//bReadyToRead :=  Tc2_System.MEMCMP( ADR( stTimeStamp), ADR (stNullTimeStamp), SIZEOF(stTimeStamp)) <> 0 AND NOT  fbGetSystemTime.BUSY;	
			(*keczi*)	(*zrobione po to zeby w wypadku jak po starcie PLC na HMI mial pokazywac czas alarmu '00:00:00', zebyb poczekal az faktycznie pokazuje date i czas*)

//Get Current System Time
fbGetSystemTime(NETID := ,
				START := bFirstScan OR bUpdateSysTime,
				TMOUT := ,
				BUSY => ,
				ERR => ,
				ERRID => ,
				TIMESTR => );
				
//Get system time done detection - one-shot
rtrigSysTimeCollected(CLK := NOT fbGetSystemTime.BUSY);

//Synchronize Real-Time clock with system time
fbRTClock(	EN := rtrigSysTimeCollected.Q, 
			PDT := fbGetSystemTime.TIMESTR,
			CDT => stTimeStamp, 
			Q => bReadyToRead);

// System Date and Time in Proper Order 
IF bReadyToRead THEN
	sRawDateTime := SYSTEMTIME_TO_STRING(stTimeStamp);  // format: YYYY-MM-DD-hh:mm:ss.xxx
	GVL_HMI_GLOBAL.sSystemDate := CONCAT(CONCAT(CONCAT(CONCAT(MID(sRawDateTime, 2, 9), '.'),  MID(sRawDateTime, 2, 6)), '.'), LEFT(sRawDateTime, 4));
	GVL_HMI_GLOBAL.sSystemTime := MID(sRawDateTime, 8, 12);
	sDateTime := CONCAT(CONCAT(GVL_HMI_GLOBAL.sSystemDate, '  '), GVL_HMI_GLOBAL.sSystemTime);
	sDateTimeSpaces	:= CONCAT(sDateTime, '    ');
END_IF;

bFirstScan := FALSE;
END_ACTION

END_PROGRAM

// ---- POUs/A_Master/PRG_MasterSystemTime.TcPOU
PROGRAM PRG_MasterSystemTime
VAR
	//Variables
	bReadyToRead				:BOOL;
	bFirstScan					:BOOL := TRUE;
	bUpdateSysTime				:BOOL; //Output of pulse generator
	tSysTimeUpdatePeriod		:TIME := T#5S;
	stTimeStamp					:TIMESTRUCT;
	stNullTimeStamp				:TIMESTRUCT;
	sRawDateTime				:STRING;
	sSystemDate					:STRING;
	sSystemTime					:STRING;
	sDateTime					:STRING;
	sDateTimeSpaces				:STRING;
	
	stTimeTest                  :TIMESTRUCT;
	sttimeTest2                 :TIMESTRUCT;
	sTestTime                   :STRING;
	nSectTest                   :DINT;
	bStartTest                  :BOOL;
	bStsrtTest2                 :BOOL;
	
	
	//Functions
	fbGetSystemTime				:TC2_Utilities.NT_GetTime;
	fbRTClock					:TC2_Utilities.RTC_EX2;		//Local real-time clock
	tonTimeUpdateGen			:TC2_Utilities.TON;			//Pulse generator for triggering fbGetSystemTime function
	rtrigSysTimeCollected		:TC2_Utilities.R_TRIG;		//System time collected

    fbTimerControl              :FB_TimeControl;
	bStartTimeTest              :BOOL;
	bResetTimeTest              :BOOL;
	nTimeHourTest               :DINT;
	nTimeMinTest                :DINT;
	nTimeSecTest                :DINT;
	nTimeTotalSecTest           :DINT;
END_VAR

//Aux functions call
tonTimeUpdateGen(	IN := NOT bUpdateSysTime,
					PT := tSysTimeUpdatePeriod,
					Q => bUpdateSysTime);

//bReadyToRead :=  Tc2_System.MEMCMP( ADR( stTimeStamp), ADR (stNullTimeStamp), SIZEOF(stTimeStamp)) <> 0 AND NOT  fbGetSystemTime.BUSY;	
			(*keczi*)	(*zrobione po to zeby w wypadku jak po starcie PLC na HMI mial pokazywac czas alarmu '00:00:00', zebyb poczekal az faktycznie pokazuje date i czas*)

//Get Current System Time
fbGetSystemTime(NETID := ,
				START := bFirstScan OR bUpdateSysTime,
				TMOUT := ,
				BUSY => ,
				ERR => ,
				ERRID => ,
				TIMESTR => );
				
//Get system time done detection - one-shot
rtrigSysTimeCollected(CLK := NOT fbGetSystemTime.BUSY);

//Synchronize Real-Time clock with system time
fbRTClock(	EN := rtrigSysTimeCollected.Q, 
			PDT := fbGetSystemTime.TIMESTR,
			CDT => stTimeStamp, 
			Q => bReadyToRead);

// System Date and Time in Proper Order 
IF bReadyToRead THEN
	sRawDateTime := SYSTEMTIME_TO_STRING(stTimeStamp);  // format: YYYY-MM-DD-hh:mm:ss.xxx
	sSystemDate := CONCAT(CONCAT(CONCAT(CONCAT(MID(sRawDateTime, 2, 9), '.'),  MID(sRawDateTime, 2, 6)), '.'), LEFT(sRawDateTime, 4));
	sSystemTime := MID(sRawDateTime, 8, 12);
	sDateTime := CONCAT(CONCAT(sSystemDate, '  '), sSystemTime);
	sDateTimeSpaces	:= CONCAT(sDateTime, '    ');
	
	//Time to write to CSV Files
	//nSystemTime := sSystemTime;
END_IF;

bFirstScan := FALSE;

IF bStartTest THEN
	sTestTime:= SYSTEMTIME_TO_STRING(stTimeTest);
END_IF

fbTimerControl( bEnable  :=  bStartTimeTest,
	            bReset   :=  bResetTimeTest,
				nHour     => nTimeHourTest,
				nMin      => nTimeMinTest,
				nSec      => nTimeSecTest,
				nTotalSec => nTimeTotalSecTest );

END_PROGRAM

// ---- POUs/E_HMI/PRG_HMI.TcPOU
PROGRAM PRG_HMI
VAR
	

	tonCaseDelay				: ARRAY [1..20] OF TON;
	tofCase						: ARRAY [1..20] OF TOF;
	rtrigCaseTriger				: ARRAY [1..20] OF R_TRIG;
	nHeightMeasureStateValue	: ARRAY [1..4] OF INT;
	i							: INT;

END_VAR

ACT_ScreensNamesSet();
ACT_Buttons();
ACT_TimTrig();
ACT_General();

ACTION ACT_Buttons:
ACT_TimTrig();

IF tonCaseDelay[1].Q THEN
	
		GVL_HMI_GLOBAL.bResetButton	:= FALSE;
		
END_IF
IF tonCaseDelay[2].Q THEN
	
		GVL_HMI_GLOBAL.bStopButton	:= FALSE;
		
END_IF
IF tonCaseDelay[3].Q THEN
	
		GVL_HMI_GLOBAL.bStartButton	:= FALSE;
		
END_IF

IF GVL_HMI_GLOBAL.bStartLeakMan THEN
	GVL_IO.dw_B07_i28General_I_O.bStart := TRUE;
END_IF
IF tonCaseDelay[4].Q THEN
	
		GVL_HMI_GLOBAL.bStartLeakMan	:= FALSE;
		GVL_IO.dw_B07_i28General_I_O.bStart := FALSE;
END_IF

IF GVL_HMI_GLOBAL.bStopLeakMan THEN
	GVL_IO.dw_B07_i28General_I_O.bStop := TRUE;
END_IF
IF tonCaseDelay[5].Q THEN
	
		GVL_HMI_GLOBAL.bStopLeakMan	:= FALSE;
		GVL_IO.dw_B07_i28General_I_O.bStop := FALSE;
		
END_IF

IF GVL_HMI_GLOBAL.bResetLeakMan THEN
	GVL_IO.dw_B07_i28General_I_O.bReset := TRUE;
END_IF
IF tonCaseDelay[6].Q THEN
	
		GVL_HMI_GLOBAL.bResetLeakMan	:= FALSE;
		GVL_IO.dw_B07_i28General_I_O.bReset := FALSE;
		
END_IF

IF tonCaseDelay[7].Q THEN
	
		GVL_HMI_GLOBAL.bShutDown	:= FALSE;
		
END_IF
IF tonCaseDelay[8].Q THEN
	
		GVL_HMI_GLOBAL.bSetLeakProgramID	:= FALSE;
		
END_IF

// Stopper Press Enable/Disable Message

IF GVL_HMI_GLOBAL.bStopperPressEnable THEN 
	GVL_HMI_GLOBAL.sStopperEnableDisable:='STOPPER PRESS ENABLED';
	ELSE
	GVL_HMI_GLOBAL.sStopperEnableDisable:='STOPPER PRESS DISABLED';
END_IF
END_ACTION

ACTION ACT_General:
IF  tofCase[1].Q
	AND (NOT GVL_MASTER.stMasterControl.bNoMachineImmediateFault OR NOT GVL_MASTER.stMasterControl.bNoCycleStopFault) THEN
	GVL_HMI_GLOBAL.bAutoCycleFaultDialog := TRUE;
END_IF
END_ACTION

ACTION ACT_ScreensNamesSet:
GVL_HMI_GLOBAL.aIOScreen[0] := 'Overview';
GVL_HMI_GLOBAL.aIOScreen[1] := 'HMI - CP2913-0000 | Beckhoff HMI';
GVL_HMI_GLOBAL.aIOScreen[2] := 'PLC - C6015-0010 | Beckhoff PLC | Windows 10 Embedded';
GVL_HMI_GLOBAL.aIOScreen[3] := 'Terminal 1- EK1100 | EtherCAT Coupler';
GVL_HMI_GLOBAL.aIOScreen[4] := 'Terminal 2 - EL6070 | Licence ';
GVL_HMI_GLOBAL.aIOScreen[5] := CONCAT('Terminal 3 - ' , GVL_IO.dw_T02_EL1809.sTerminalName);
GVL_HMI_GLOBAL.aIOScreen[6] := CONCAT('Terminal 4 - ' , GVL_IO.dw_T03_EL2809.sTerminalName);
GVL_HMI_GLOBAL.aIOScreen[7] := 'Terminal 12 - EL6631 |  2-port communication interface';
GVL_HMI_GLOBAL.aIOScreen[8] := 'I28 | Cincinnati Leak Tester | ProfiNET';

GVL_HMI_GLOBAL.aManualScreen[0] := 'Cognex | Vision Test';
GVL_HMI_GLOBAL.aManualScreen[1] := 'Keyence | Height Test';
GVL_HMI_GLOBAL.aManualScreen[2] := 'Cincinnati | Leak Test';
END_ACTION

ACTION ACT_TimTrig:


tonCaseDelay[1](IN:= GVL_HMI_GLOBAL.bResetButton,PT:=T#500MS);
tonCaseDelay[2](IN:= GVL_HMI_GLOBAL.bStopButton,PT:=T#500MS);
tonCaseDelay[3](IN:= GVL_HMI_GLOBAL.bStartButton,PT:=T#500MS);
tonCaseDelay[4](IN:= GVL_HMI_GLOBAL.bStartLeakMan,PT:=T#500MS);
tonCaseDelay[5](IN:= GVL_HMI_GLOBAL.bStopLeakMan,PT:=T#500MS);
tonCaseDelay[6](IN:= GVL_HMI_GLOBAL.bResetLeakMan,PT:=T#500MS);
//tonCaseDelay[7](IN:= GVL_HMI_GLOBAL.bShutDown,PT:=T#500MS);
tonCaseDelay[8](IN:= GVL_HMI_GLOBAL.bSetLeakProgramID,PT:=T#5S);
tonCaseDelay[9](IN:= ,PT:=T#1S);
tonCaseDelay[10](IN:= ,PT:=T#1S);

tofCase[1](IN:= GVL_MASTER.stStationSruct[0].nState > 1000 AND GVL_MASTER.stStationSruct[0].nState < 1900,PT:=T#1S);



rtrigCaseTriger[1](CLK := GVL_MASTER.stNest.bPieceReject);
END_ACTION

END_PROGRAM

// ---- POUs/G_Utility/PRG_Puls.TcPOU
PROGRAM PRG_Puls
VAR
    //=== Master Pulses ===//
	fbScalingFlash  :FB_Pulse;
	fbScalingFlash4 :FB_Pulse;
	fbScalingFlash5 :FB_Pulse;
	fbFlash100Hz    :FB_Pulse;
	fbFlash10Hz		:FB_Pulse;
	fbFlash10HzB    :FB_Pulse;
	fbFlash4Hz		:FB_Pulse;
	fbFlash2Hz		:FB_Pulse;
	fbFlash1Hz		:FB_Pulse;			

END_VAR

    //=== Master Pulses ===//
(**************************************************************************************************)
fbScalingFlash(
	bEnable	:=	TRUE,
	tPulseOn	:=	T#2MS,
	tPulseOff	:=	T#2MS,
	bFlash		=>	GVL_MASTER.bFlashScale
);

fbScalingFlash4(
     bEnable	:=	TRUE,
	tPulseOn	:=	T#4MS,
	tPulseOff	:=	T#4MS,
	bFlash		=>	GVL_MASTER.bFlashScale4
);
fbScalingFlash5(
     bEnable	:=	TRUE,
	tPulseOn	:=	T#5MS,
	tPulseOff	:=	T#5MS,
	bFlash		=>	GVL_MASTER.bFlashScale5
);



fbFlash100Hz(
	bEnable	:=	TRUE,
	tPulseOn	:=	T#10MS,
	tPulseOff	:=	T#10MS,
	bFlash		=>	GVL_MASTER.bFlash100Hz
);


fbFlash10HzB ( 
    bEnable	    :=	TRUE,
	tPulseOn	:=	T#20MS,//  T#50MS,
	tPulseOff	:=	T#20MS,//  T#50MS,
	bFlash		=>	GVL_MASTER.bFlash10BHz
);


fbFlash10Hz(
	bEnable	:=	TRUE,
	tPulseOn	:=	T#100MS,
	tPulseOff	:=	T#100MS,
	bFlash		=>	GVL_MASTER.bFlash10Hz
);


fbFlash4Hz(
	bEnable	:=	TRUE,
	tPulseOn	:=	T#250MS,
	tPulseOff	:=	T#250MS,
	bFlash		=>	GVL_MASTER.bFlash4Hz
);

fbFlash2Hz(
	bEnable	:=	TRUE,
	tPulseOn	:=	T#500MS,
	tPulseOff	:=	T#500MS,
	bFlash		=>	GVL_MASTER.bFlash2Hz
);

fbFlash1Hz(
	bEnable	:=	TRUE,
	tPulseOn	:=	T#1000MS,
	tPulseOff	:=	T#1000MS,
	bFlash		=>	GVL_MASTER.bFlash1Hz
);

END_PROGRAM

// ---- POUs/A_Master/PRG_TerminBoxInfo.TcPOU
PROGRAM PRG_TerminBoxInfo
VAR
END_VAR

//Terminal 0
GVL_IO.dwTerminalInfo[1].fbTerminalInfo(nTerminalState:= 8,
                                        sTerminalState => GVL_IO.dwTerminalInfo[0].sTerminalInfo);
//Terminal 1
GVL_IO.dwTerminalInfo[1].fbTerminalInfo(nTerminalState:= GVL_IO.dwTerminalInfo[1].nTerminal_State,
                                        sTerminalState => GVL_IO.dwTerminalInfo[1].sTerminalInfo);  
//Terminal 2
GVL_IO.dwTerminalInfo[2].fbTerminalInfo(nTerminalState:= GVL_IO.dwTerminalInfo[2].nTerminal_State,
                                        sTerminalState => GVL_IO.dwTerminalInfo[2].sTerminalInfo); 
//Terminal 3
GVL_IO.dwTerminalInfo[3].fbTerminalInfo(nTerminalState:= GVL_IO.dwTerminalInfo[3].nTerminal_State,
                                        sTerminalState => GVL_IO.dwTerminalInfo[3].sTerminalInfo); 
//Terminal 4
GVL_IO.dwTerminalInfo[4].fbTerminalInfo(nTerminalState:= GVL_IO.dwTerminalInfo[4].nTerminal_State,
                                        sTerminalState => GVL_IO.dwTerminalInfo[4].sTerminalInfo); 
//Terminal 5
GVL_IO.dwTerminalInfo[5].fbTerminalInfo(nTerminalState:= GVL_IO.dwTerminalInfo[5].nTerminal_State,
                                        sTerminalState => GVL_IO.dwTerminalInfo[5].sTerminalInfo); 
//Terminal 6
GVL_IO.dwTerminalInfo[6].fbTerminalInfo(nTerminalState:= GVL_IO.dwTerminalInfo[6].nTerminal_State,
                                        sTerminalState => GVL_IO.dwTerminalInfo[6].sTerminalInfo); 
//Terminal 7
GVL_IO.dwTerminalInfo[7].fbTerminalInfo(nTerminalState:= GVL_IO.dwTerminalInfo[7].nTerminal_State,
                                        sTerminalState => GVL_IO.dwTerminalInfo[7].sTerminalInfo); 
//Terminal 8
GVL_IO.dwTerminalInfo[8].fbTerminalInfo(nTerminalState:= GVL_IO.dwTerminalInfo[8].nTerminal_State,
                                        sTerminalState => GVL_IO.dwTerminalInfo[8].sTerminalInfo); 
//Terminal 9
GVL_IO.dwTerminalInfo[9].fbTerminalInfo(nTerminalState:= GVL_IO.dwTerminalInfo[9].nTerminal_State,
                                        sTerminalState => GVL_IO.dwTerminalInfo[9].sTerminalInfo); 
//Terminal 10
GVL_IO.dwTerminalInfo[10].fbTerminalInfo(nTerminalState:= GVL_IO.dwTerminalInfo[10].nTerminal_State,
                                        sTerminalState => GVL_IO.dwTerminalInfo[10].sTerminalInfo); 
//Terminal 11
GVL_IO.dwTerminalInfo[11].fbTerminalInfo(nTerminalState:= GVL_IO.dwTerminalInfo[11].nTerminal_State,
                                        sTerminalState => GVL_IO.dwTerminalInfo[11].sTerminalInfo); 
//Terminal 12
GVL_IO.dwTerminalInfo[12].fbTerminalInfo(nTerminalState:= GVL_IO.dwTerminalInfo[12].nTerminal_State,
                                        sTerminalState => GVL_IO.dwTerminalInfo[12].sTerminalInfo); 										
//Terminal 13
GVL_IO.dwTerminalInfo[13].fbTerminalInfo(nTerminalState:= GVL_IO.dwTerminalInfo[13].nTerminal_State,
                                        sTerminalState => GVL_IO.dwTerminalInfo[13].sTerminalInfo); 
//Terminal 14
GVL_IO.dwTerminalInfo[14].fbTerminalInfo(nTerminalState:= GVL_IO.dwTerminalInfo[14].nTerminal_State,
                                        sTerminalState => GVL_IO.dwTerminalInfo[14].sTerminalInfo);
										
//Terminal 15
GVL_IO.dwTerminalInfo[15].fbTerminalInfo(nTerminalState:= GVL_IO.dwTerminalInfo[15].nTerminal_State,
                                        sTerminalState => GVL_IO.dwTerminalInfo[15].sTerminalInfo); 
//Terminal 16
GVL_IO.dwTerminalInfo[16].fbTerminalInfo(nTerminalState:= 8,
                                        sTerminalState => GVL_IO.dwTerminalInfo[16].sTerminalInfo);										

//Terminal 17
GVL_IO.dwTerminalInfo[17].fbTerminalInfo(nTerminalState:= 8,
                                        sTerminalState => GVL_IO.dwTerminalInfo[17].sTerminalInfo);

//Terminal 18
GVL_IO.dwTerminalInfo[18].fbTerminalInfo(nTerminalState:= 8,
                                        sTerminalState => GVL_IO.dwTerminalInfo[18].sTerminalInfo);

//Terminal 19
GVL_IO.dwTerminalInfo[19].fbTerminalInfo(nTerminalState:= 8,
                                        sTerminalState => GVL_IO.dwTerminalInfo[19].sTerminalInfo);

//Terminal 20
GVL_IO.dwTerminalInfo[20].fbTerminalInfo(nTerminalState:= 8,
                                        sTerminalState => GVL_IO.dwTerminalInfo[20].sTerminalInfo);
																				
// Box 15
GVL_IO.dwBoxInfo[15].fbBoxInfo(nPnIoBoxState := GVL_IO.dwBoxInfo[15].nPnIoBoxState,    	
                               nPnIoBoxDiag  := GVL_IO.dwBoxInfo[15].nPnIoBoxDiag,
							   sBoxState      => GVL_IO.dwBoxInfo[15].sBoxState,
                               sBoxDiag       => GVL_IO.dwBoxInfo[15].sBoxDiag);
							   
//===========================================================================================================

END_PROGRAM

// ---- POUs/C_LeakTest/PRG_LeakTestEvents_Info.TcPOU
PROGRAM PRG_LeakTestEvents_Info
VAR
	
	asLeakTesterSegments 				: ARRAY [0..200] OF WSTRING;
	asLeakTesterTestData 				: ARRAY [0..200] OF WSTRING;
	asLeakTesterUnit 	 				: ARRAY [0..200] OF WSTRING;
	asLeakTesterPrecision				: ARRAY [0..10]  OF WSTRING;
	asLeakTesterProgramEvaluation		: ARRAY [0..20]  OF WSTRING;
	asLeakTesterTestEvaluation			: ARRAY [0..150]  OF WSTRING;
	asLeakTesterTestType				: ARRAY [0..25]  OF WSTRING;
	fLeakTesterActive					: F_TRIG;
	bLeakTesterActive					: BOOL;
	Test1								: BOOL;
		
	i									: DINT;
	

END_VAR

ACT_LiveSegmentCode();
ACT_LeakTesterTestData();
ACT_LeakTesterUnit();
ACT_Precision();
ACT_ProgramEvaluation();
ACT_LeakTesterTestEvaluation();
ACT_TestType();

//Last Result DATA

GVL_IO.dw_B07_i28LastResult.sPartEvaluation 		:= asLeakTesterTestData[GVL_IO.dw_B07_i28LastResult.inTestType];
GVL_IO.dw_B07_i28LastResult.sPrecision				:= asLeakTesterPrecision[GVL_IO.dw_B07_i28LastResult.inPrecisionCode];
GVL_IO.dw_B07_i28LastResult.sTestType				:= asLeakTesterTestType[ GVL_IO.dw_B07_i28LastResult.inPartEvaluation];
GVL_IO.dw_B07_i28LastResult.sUnit1      			:= asLeakTesterUnit[GVL_IO.dw_B07_i28LastResult.inUnitCode1];
GVL_IO.dw_B07_i28LastResult.sUnit2					:= asLeakTesterUnit[GVL_IO.dw_B07_i28LastResult.inUnitCode2];
GVL_IO.dw_B07_i28LastResult.sVariable1				:= asLeakTesterTestData[GVL_IO.dw_B07_i28LastResult.inVariableCode1];
GVL_IO.dw_B07_i28LastResult.sVariable2				:= asLeakTesterTestData[GVL_IO.dw_B07_i28LastResult.inVariableCode2];

//Live DATA


GVL_IO.dw_B07_i28LiveMeasurement.sPrecision1		:= asLeakTesterPrecision[GVL_IO.dw_B07_i28LiveMeasurement.inPrecisionCode1];
GVL_IO.dw_B07_i28LiveMeasurement.sPrecision2		:= asLeakTesterPrecision[GVL_IO.dw_B07_i28LiveMeasurement.inPrecisionCode2];
GVL_IO.dw_B07_i28LiveMeasurement.sPrecision3		:= asLeakTesterPrecision[GVL_IO.dw_B07_i28LiveMeasurement.inPrecisionCode3];
GVL_IO.dw_B07_i28LiveMeasurement.sPrecision4		:= asLeakTesterPrecision[GVL_IO.dw_B07_i28LiveMeasurement.inPrecisionCode4];
GVL_IO.dw_B07_i28LiveMeasurement.sSegmentCode		:= asLeakTesterSegments[GVL_IO.dw_B07_i28LiveMeasurement.inSegmentCode];
GVL_IO.dw_B07_i28LiveMeasurement.sUnit1				:= asLeakTesterUnit[GVL_IO.dw_B07_i28LiveMeasureMENT.inUnitCode1];
GVL_IO.dw_B07_i28LiveMeasurement.sUnit2				:= asLeakTesterUnit[GVL_IO.dw_B07_i28LiveMeasureMENT.inUnitCode2];
GVL_IO.dw_B07_i28LiveMeasurement.sUnit3				:= asLeakTesterUnit[GVL_IO.dw_B07_i28LiveMeasureMENT.inUnitCode3];
GVL_IO.dw_B07_i28LiveMeasurement.sUnit4				:= asLeakTesterUnit[GVL_IO.dw_B07_i28LiveMeasureMENT.inUnitCode4];
GVL_IO.dw_B07_i28LiveMeasurement.sVariable1			:= asLeakTesterTestData[GVL_IO.dw_B07_i28LiveMeasurement.inVariableCode1];
GVL_IO.dw_B07_i28LiveMeasurement.sVariable2			:= asLeakTesterTestData[GVL_IO.dw_B07_i28LiveMeasurement.inVariableCode2];
GVL_IO.dw_B07_i28LiveMeasurement.sVariable3			:= asLeakTesterTestData[GVL_IO.dw_B07_i28LiveMeasurement.inVariableCode3];
GVL_IO.dw_B07_i28LiveMeasurement.sVariable4			:= asLeakTesterTestData[GVL_IO.dw_B07_i28LiveMeasurement.inVariableCode4];


ACT_LastResultSet();

ACTION ACT_LastResultSet:

fLeakTesterActive(CLK := GVL_IO.dw_B07_i28General_I_O.bTestActiveLiveData, Q => bLeakTesterActive);


IF bLeakTesterActive THEN
	
	FOR i :=200 TO 1 BY (-1) DO
		GVL_PERSIST.ast_i28LasResult[i]	:= GVL_PERSIST.ast_i28LasResult[i-1];
	END_FOR
	
	GVL_PERSIST.ast_i28LasResult[0] := GVL_IO.dw_B07_i28LastResult;
	GVL_PERSIST.ast_i28LasResult[0].sTime := GVL_HMI_GLOBAL.sSystemTime;
	GVL_PERSIST.ast_i28LasResult[0].sDate := GVL_HMI_GLOBAL.sSystemDate;

END_IF
END_ACTION

ACTION ACT_LeakTesterTestData:
asLeakTesterTestData[0] := "NO DATA";
asLeakTesterTestData[1] := "Elapsed Timer";
asLeakTesterTestData[2] := "Segment Timer";
asLeakTesterTestData[3] := "Test Execution Time";
asLeakTesterTestData[4] := "Target Pressure";
asLeakTesterTestData[5] := "Test Pressure";
asLeakTesterTestData[6] := "Master Part Profile Test Pressure";
asLeakTesterTestData[7] := "Master Part & Leak Profile Test Pressure";
asLeakTesterTestData[8] := "Leak Standard Calibrated Pressure";
asLeakTesterTestData[9] := "Self Test Pressure";
asLeakTesterTestData[10] := "Measured Pressure";
asLeakTesterTestData[11] := "Instrument Pressure";
asLeakTesterTestData[12] := "Master Gauge Pressure";
asLeakTesterTestData[13] := "Master Part Pressure Loss (Corrected)";
asLeakTesterTestData[14] := "Low Limit Pressure Loss";
asLeakTesterTestData[15] := "High Limit Pressure Loss";
asLeakTesterTestData[16] := "Master Part & Leak Pressure Loss (Corrected)";
asLeakTesterTestData[17] := "Pressure Loss (Corrected)";
asLeakTesterTestData[18] := "Pressure Loss (Actual Read)";
asLeakTesterTestData[19] := "Master Part Flow Offset (Corrected)";
asLeakTesterTestData[20] := "Performance Factor";
asLeakTesterTestData[21] := "Low Limit Rate";
asLeakTesterTestData[22] := "High Limit Rate";
asLeakTesterTestData[23] := "Loss Rate (Corrected)";
asLeakTesterTestData[24] := "Loss Rate (Actual Read)";
asLeakTesterTestData[25] := "Quik Test Pressure";
asLeakTesterTestData[26] := "Quik Test Loss (Corrected)";
asLeakTesterTestData[27] := "Quik Test Flow (Corrected)";
asLeakTesterTestData[28] := "Low Limit Leak Rate";
asLeakTesterTestData[29] := "High Limit Leak Rate";
asLeakTesterTestData[30] := "Predicted Leak Rate";
asLeakTesterTestData[31] := "Leak Rate";
asLeakTesterTestData[32] := "Corrected Leak Standard Calibrated Flow";
asLeakTesterTestData[33] := "Measured Flow";
asLeakTesterTestData[34] := "Environmental Drift Correction Offset";
asLeakTesterTestData[35] := "Transducer Type";
asLeakTesterTestData[36] := "Transducer Typical Residual";
asLeakTesterTestData[37] := "Transducer Zero Low Window";
asLeakTesterTestData[38] := "Transducer Zero High Window";
asLeakTesterTestData[39] := "Regulator Type";
asLeakTesterTestData[40] := "Analog A/D Value";
asLeakTesterTestData[41] := "Peak Pressure";
asLeakTesterTestData[42] := "Analog Input";
asLeakTesterTestData[43] := "Analog Output";
asLeakTesterTestData[44] := "Event Delta Pressure";
asLeakTesterTestData[45] := "Alternate Leak Rate";
asLeakTesterTestData[46] := "DP Master Part Pressure Loss (Corrected)";
asLeakTesterTestData[47] := "DP Master Part & Leak Pressure Loss (Corrected)";
asLeakTesterTestData[48] := "Master Part Quik Pressure Loss (Corrected)";
asLeakTesterTestData[49] := "Master Part Quik Pressure Loss (Actual Read)";
asLeakTesterTestData[50] := "Master Part & Leak Quik Pressure Loss (Corrected)";
asLeakTesterTestData[51] := "Master Part & Leak Quik Pressure Loss (Actual Read)";
asLeakTesterTestData[52] := "Master Part Quik Test Pressure";
asLeakTesterTestData[53] := "Master Part & Leak Quik Test Pressure";
asLeakTesterTestData[54] := "Master Part Quik DP Pressure Loss (Corrected)";
asLeakTesterTestData[55] := "Master Part Quik DP Pressure Loss (Actual Read)";
asLeakTesterTestData[56] := "Master Part & Leak Quik DP Pressure Loss (Actual Read)";
asLeakTesterTestData[57] := "Signal to Noise Ratio";
asLeakTesterTestData[58] := "Effective Number of Bits";
asLeakTesterTestData[59] := "Flicker Free Number of Bits";
asLeakTesterTestData[60] := "High Limit Percent Volume";
asLeakTesterTestData[61] := "Part Percent Volume";
asLeakTesterTestData[62] := "Reference Pressure";
asLeakTesterTestData[63] := "Fill Pressure";
asLeakTesterTestData[64] := "Transducer Cal/Verify - Number of Points";
asLeakTesterTestData[65] := "Transducer - Setpoint Pressure Value";
asLeakTesterTestData[66] := "Transducer - Instrument Pressure Reading";
asLeakTesterTestData[67] := "Transducer - Instrument Flow Reading";
asLeakTesterTestData[68] := "Transducer - Analog Value";
asLeakTesterTestData[69] := "Transducer - Master Reading";
asLeakTesterTestData[70] := "Transducer - Master Value";
asLeakTesterTestData[71] := "Transducer - Atmospheric Pressure";
asLeakTesterTestData[72] := "Transducer - Linearity";
asLeakTesterTestData[73] := "Electronic Regulator Cal - Number of Points";
asLeakTesterTestData[74] := "Electronic Regulator - Instrument Pressure Reading";
asLeakTesterTestData[75] := "Electronic Regulator - Analog Value";
asLeakTesterTestData[76] := "Electronic Regulator - Master Value";
asLeakTesterTestData[77] := "Electronic Regulator Analysis - Number of Points";
asLeakTesterTestData[78] := "Electronic Regulator Analysis - Instrument Pressure Reading";
asLeakTesterTestData[79] := "Electronic Regulator Analysis - Voltage Low Limit";
asLeakTesterTestData[80] := "Electronic Regulator Analysis - Voltage High Limit";
asLeakTesterTestData[81] := "Event Pressure";
asLeakTesterTestData[82] := "Part Flow";
asLeakTesterTestData[83] := "Pre-Pressure";
asLeakTesterTestData[84] := "Tracer Cumulative Leak Rate";
asLeakTesterTestData[85] := "Sniffer Test Location";
asLeakTesterTestData[86] := "Electronic Regulator Cal - Atmospheric Pressure";
asLeakTesterTestData[87] := "REF External Xdcr Pressure";
asLeakTesterTestData[88] := "Differential Pressure Loss (Corrected)";
asLeakTesterTestData[89] := "Differential Pressure Loss (Actual Read)";
asLeakTesterTestData[90] := "Reference Pressure Loss";
asLeakTesterTestData[91] := "Differential Pressure Loss (Actual Read)";
asLeakTesterTestData[92] := "Input State";
asLeakTesterTestData[93] := "Leak Loss";
asLeakTesterTestData[94] := "Batch Quantity";
asLeakTesterTestData[95] := "DP Leak Loss";
asLeakTesterTestData[96] := "Average Quantity";
asLeakTesterTestData[97] := "Charge Pressure";
asLeakTesterTestData[98] := "Standard Pressure";
asLeakTesterTestData[99] := "Instrument Volume";
asLeakTesterTestData[100] := "Part Volume";
asLeakTesterTestData[101] := "Test Measurement Time";
asLeakTesterTestData[102] := "Calculated Leak Rate Offset";
END_ACTION

ACTION ACT_LeakTesterTestEvaluation:
asLeakTesterTestEvaluation[0] := "NO DATA";
asLeakTesterTestEvaluation[1] := "PROGRAM ACCEPT";
asLeakTesterTestEvaluation[2] := "PROGRAM REJECT";
asLeakTesterTestEvaluation[3] := "PART REJECT - LEVEL 1";
asLeakTesterTestEvaluation[4] := "PART REJECT - LEVEL 2";
asLeakTesterTestEvaluation[5] := "PART REJECT - LEVEL 3";
asLeakTesterTestEvaluation[6] := "PROGRAM CALIBRATION PASSED";
asLeakTesterTestEvaluation[7] := "PROGRAM CALIBRATION FAILED";
asLeakTesterTestEvaluation[8] := "MASTER PART COMPLETE";
asLeakTesterTestEvaluation[9] := "SELF-TEST PASSED";
asLeakTesterTestEvaluation[10] := "SELF-TEST FAILED";
asLeakTesterTestEvaluation[11] := "SEQUENCE COMPLETE";
asLeakTesterTestEvaluation[12] := "SEVERE LEAK";
asLeakTesterTestEvaluation[13] := "TEST PRESSURE LOW";
asLeakTesterTestEvaluation[14] := "TEST PRESSURE HIGH";
asLeakTesterTestEvaluation[15] := "BELOW TARGET PRESSURE";
asLeakTesterTestEvaluation[16] := "ABOVE TARGET PRESSURE";
asLeakTesterTestEvaluation[17] := "HELIUM BACKGROUND FAULT";
asLeakTesterTestEvaluation[18] := "PART EVAC FAULT";
asLeakTesterTestEvaluation[19] := "TRANSDUCER ZERO BAD";
asLeakTesterTestEvaluation[20] := "TRANSDUCER OVER-RANGE";
asLeakTesterTestEvaluation[21] := "FLOW TRANSDUCER ZERO BAD";
asLeakTesterTestEvaluation[22] := "FLOW TRANSDUCER OVER-RANGE";
asLeakTesterTestEvaluation[23] := "ERROR: EXCESSIVE FLOW";
asLeakTesterTestEvaluation[24] := "PROGRAM CONFIGURATION ERROR";
asLeakTesterTestEvaluation[25] := "PROG ERROR";
asLeakTesterTestEvaluation[26] := "CALCULATION ERROR";
asLeakTesterTestEvaluation[27] := "INVALID PROGRAM SELECTED";
asLeakTesterTestEvaluation[28] := "INVALID CALIBRATION DATA";
asLeakTesterTestEvaluation[29] := "INVALID I/O CONFIGURATION";
asLeakTesterTestEvaluation[30] := "I/O FAULT";
asLeakTesterTestEvaluation[31] := "CAL REQUIRED - LIMIT EXCEEDED";
asLeakTesterTestEvaluation[32] := "CAL REQUIRED - PARAM CHANGED";
asLeakTesterTestEvaluation[33] := "MIN PERF FACTOR ERROR";
asLeakTesterTestEvaluation[34] := "MASTER+LEAK LOSS<MASTER LOSS";
asLeakTesterTestEvaluation[35] := "MASTER LOSS>MAX M+L LOSS";
asLeakTesterTestEvaluation[36] := "MASTER+LEAK LOSS>MAX M+L LOSS";
asLeakTesterTestEvaluation[37] := "MASTER FLOW>MAX M+L FLOW";
asLeakTesterTestEvaluation[38] := "MASTER FLOW<MIN MASTER FLOW";
asLeakTesterTestEvaluation[39] := "MASTER+LEAK FLOW>MAX M+L FLOW";
asLeakTesterTestEvaluation[40] := "MASTER FLOW>MAX MASTER FLOW";
asLeakTesterTestEvaluation[41] := "MASTER+LEAK FLOW>MAX MASTER FLOW";
asLeakTesterTestEvaluation[42] := "MASTER LOSS<MIN MASTER LOSS";
asLeakTesterTestEvaluation[43] := "MASTER LOSS>MAX MASTER LOSS";
asLeakTesterTestEvaluation[44] := "STOP BUTTON PRESSED";
asLeakTesterTestEvaluation[45] := "STOP INPUT RECEIVED";
asLeakTesterTestEvaluation[46] := "ERROR: STOP INPUT HIGH";
asLeakTesterTestEvaluation[47] := "START COMMON INPUT LOW";
asLeakTesterTestEvaluation[48] := "ERROR: ANTI-TIE DOWN";
asLeakTesterTestEvaluation[49] := "ERROR: PART NOT PRESENT";
asLeakTesterTestEvaluation[50] := "ERROR: PART NOT CHANGED";
asLeakTesterTestEvaluation[51] := "EXT SWITCH DID NOT GO LOW";
asLeakTesterTestEvaluation[52] := "EXT SWITCH DID NOT GO HIGH";
asLeakTesterTestEvaluation[53] := "ERROR: TOOLING NOT RESET";
asLeakTesterTestEvaluation[54] := "ERROR: TOOLING NOT EXTENDED";
asLeakTesterTestEvaluation[55] := "ERROR: TOOLING NOT RETRACTED";
asLeakTesterTestEvaluation[56] := "TOOLING RESET";
asLeakTesterTestEvaluation[57] := "ERROR: PART MARK FAULT";
asLeakTesterTestEvaluation[58] := "PART NOT FULL";
asLeakTesterTestEvaluation[59] := "PART NOT EXHAUSTED";
asLeakTesterTestEvaluation[60] := "PART NOT STABILIZED";
asLeakTesterTestEvaluation[61] := "AUTOSETUP SEQ COMPLETE";
asLeakTesterTestEvaluation[62] := "DP TRANSDUCER ZERO BAD";
asLeakTesterTestEvaluation[63] := "DP TRANSDUCER OVER-RANGE";
asLeakTesterTestEvaluation[64] := "ERROR: TWO-INPUT REQ TO START";
asLeakTesterTestEvaluation[65] := "ERROR: BARCODE REQ TO START";
asLeakTesterTestEvaluation[66] := "DP TRANSDUCER FAULT";
asLeakTesterTestEvaluation[67] := "ERROR: NO LINKS DEFINED";
asLeakTesterTestEvaluation[68] := "ERROR: LINK EXECUTION LOOP";
asLeakTesterTestEvaluation[69] := "ERROR: LINK PROG IS PARENT";
asLeakTesterTestEvaluation[70] := "ERROR: LINK PROG UNDEFINED";
asLeakTesterTestEvaluation[71] := "ERROR: DISSIMILAR LINK ORDER";
asLeakTesterTestEvaluation[72] := "ERROR: DUPLICATE TARGET LINK";
asLeakTesterTestEvaluation[73] := "CAL PROGRAM ACCEPT";
asLeakTesterTestEvaluation[74] := "CAL PROGRAM REJECT";
asLeakTesterTestEvaluation[75] := "PRESSURE TRANSDUCER FAULT";
asLeakTesterTestEvaluation[76] := "NO EVENT OCCURRED";
asLeakTesterTestEvaluation[77] := "SYSTEM PRESSURE EXCEEDED";
asLeakTesterTestEvaluation[78] := "PRESSURE SELECT CONFIG ERROR";
asLeakTesterTestEvaluation[79] := "LEAK STD SELECT CONFIG ERROR";
asLeakTesterTestEvaluation[80] := "VENT PART RESET TOOLING";
asLeakTesterTestEvaluation[81] := "TRANSDUCER CAL COMPLETE";
asLeakTesterTestEvaluation[82] := "TRANSDUCER CAL ERROR";
asLeakTesterTestEvaluation[83] := "TRANSDUCER VERIFY COMPLETE";
asLeakTesterTestEvaluation[84] := "ELEC REGULATOR CAL COMPLETE";
asLeakTesterTestEvaluation[85] := "ELEC REGULATOR CAL ERROR";
asLeakTesterTestEvaluation[86] := "SYSTEM ERROR - SERVICE REQ";
asLeakTesterTestEvaluation[87] := "TEST PORT SELECT CONFIG ERROR";
asLeakTesterTestEvaluation[88] := "SOURCE PRESSURE EXCEEDED";
asLeakTesterTestEvaluation[89] := "PRE-PRESSURE LOW";
asLeakTesterTestEvaluation[90] := "PRE-PRESSURE HIGH";
asLeakTesterTestEvaluation[91] := "ERROR: SNIFFER NOT READY";
asLeakTesterTestEvaluation[92] := "SNIFFER UNITS MISMATCH";
asLeakTesterTestEvaluation[93] := "SNIFFER MODE MISMATCH";
asLeakTesterTestEvaluation[94] := "T-GAS BACKGROUND FAULT";
asLeakTesterTestEvaluation[95] := "T-GAS MIN LEAK RATE FAULT";
asLeakTesterTestEvaluation[96] := "T-GAS CHAMBER CLEANUP FAULT";
asLeakTesterTestEvaluation[97] := "SNIFFER TYPE MISMATCH";
asLeakTesterTestEvaluation[98] := "SNIFFER READY INPUT FAULT";
asLeakTesterTestEvaluation[99] := "CHAMBER EVACUATION FAULT";
asLeakTesterTestEvaluation[100] := "CHAMBER RISE FAULT";
asLeakTesterTestEvaluation[101] := "SCALE CONFIG ERROR";
asLeakTesterTestEvaluation[102] := "SCALE NOT READY";
asLeakTesterTestEvaluation[103] := "SCALE NOT STABLE";
asLeakTesterTestEvaluation[104] := "SCALE WEIGHT LOW";
asLeakTesterTestEvaluation[105] := "SCALE WEIGHT HIGH";
asLeakTesterTestEvaluation[106] := "WEIGHT BELOW MIN";
asLeakTesterTestEvaluation[107] := "WEIGHT ABOVE MAX";
asLeakTesterTestEvaluation[108] := "ATMOSPHERIC PRESSURE COMPLETE";
asLeakTesterTestEvaluation[109] := "ATMOSPHERIC PRESSURE ERROR";
asLeakTesterTestEvaluation[110] := "EXTERNAL XDCR PRESS";
asLeakTesterTestEvaluation[111] := "MAN FILL SWITCH";
asLeakTesterTestEvaluation[112] := "ISOLATION FAILURE";
asLeakTesterTestEvaluation[113] := "LD ZERO < MIN";
asLeakTesterTestEvaluation[114] := "LD ZERO > MAX";
asLeakTesterTestEvaluation[115] := "LD LEAK < MIN";
asLeakTesterTestEvaluation[116] := "LD LEAK > MAX";
asLeakTesterTestEvaluation[117] := "PROCESS FAULT";
asLeakTesterTestEvaluation[118] := "POWER RESET";
asLeakTesterTestEvaluation[119] := "INVALID INPUT CONFIGURATION";
asLeakTesterTestEvaluation[120] := "INPUT INITIAL STATE ERROR";
asLeakTesterTestEvaluation[121] := "MASS SPEC CONTAMINATION";
asLeakTesterTestEvaluation[122] := "CHAMBER PRESSURE HIGH";
asLeakTesterTestEvaluation[123] := "CHAMBER CROSSOVER INPUT FAULT";
asLeakTesterTestEvaluation[124] := "CHAMBER RISE INPUT FAULT";
asLeakTesterTestEvaluation[125] := "T-GAS PART FILL FAULT";
asLeakTesterTestEvaluation[126] := "T-GAS LEAK STD FAULT";
asLeakTesterTestEvaluation[127] := "MASTER+LEAK LOSS<MIN M+L LOSS";
asLeakTesterTestEvaluation[128] := "LEAK LOSS<MIN LEAK LOSS";
asLeakTesterTestEvaluation[129] := "LEAK LOSS>MAX LEAK LOSS";
asLeakTesterTestEvaluation[130] := "MASTER+LEAK FLOW<MIN M+L FLOW";
asLeakTesterTestEvaluation[131] := "LEAK FLOW<MIN LEAK FLOW";
asLeakTesterTestEvaluation[132] := "LEAK FLOW > MAX LEAK FLOW";
asLeakTesterTestEvaluation[133] := "MASTER+LEAK PART COMPLETE";
asLeakTesterTestEvaluation[134] := "VALVE LOAD FAULT";
asLeakTesterTestEvaluation[135] := "ERROR: INSTRUMENT NOT ENABLED";
asLeakTesterTestEvaluation[136] := "CHARGE PRESSURE LOW";
asLeakTesterTestEvaluation[137] := "CHARGE PRESSURE HIGH";
END_ACTION

ACTION ACT_LeakTesterUnit:
asLeakTesterUnit[0] := "NO DATA";
asLeakTesterUnit[1] := "atm";
asLeakTesterUnit[2] := "bar";
asLeakTesterUnit[3] := "cmHg";
asLeakTesterUnit[4] := "inHg";
asLeakTesterUnit[5] := "kPa";
asLeakTesterUnit[6] := "MPa";
asLeakTesterUnit[7] := "mbar";
asLeakTesterUnit[8] := "mmHg";
asLeakTesterUnit[9] := "Pa";
asLeakTesterUnit[10] := "Torr";
asLeakTesterUnit[11] := "psig";
asLeakTesterUnit[12] := "psiv";
asLeakTesterUnit[13] := "iWC";
asLeakTesterUnit[14] := "cmWC";
asLeakTesterUnit[15] := "mmWC";
asLeakTesterUnit[16] := "ksc";
asLeakTesterUnit[17] := "psia";
asLeakTesterUnit[18] := "datm";
asLeakTesterUnit[19] := "dbar";
asLeakTesterUnit[20] := "dcmHg";
asLeakTesterUnit[21] := "dinHg";
asLeakTesterUnit[22] := "dkPa";
asLeakTesterUnit[23] := "dMpa";
asLeakTesterUnit[24] := "dmbar";
asLeakTesterUnit[25] := "dmmHg";
asLeakTesterUnit[26] := "dPa";
asLeakTesterUnit[27] := "dTorr";
asLeakTesterUnit[28] := "dpsig";
asLeakTesterUnit[29] := "dpsiv";
asLeakTesterUnit[30] := "diWC";
asLeakTesterUnit[31] := "dcmWC";
asLeakTesterUnit[32] := "dmmWC";
asLeakTesterUnit[33] := "dksc";
asLeakTesterUnit[34] := "dpsi";
asLeakTesterUnit[35] := "sccm";
asLeakTesterUnit[36] := "sces";
asLeakTesterUnit[37] := "scch";
asLeakTesterUnit[38] := "scfm";
asLeakTesterUnit[39] := "slpm";
asLeakTesterUnit[40] := "slps";
asLeakTesterUnit[41] := "scfh";
asLeakTesterUnit[42] := "scfs";
asLeakTesterUnit[43] := "slph";
asLeakTesterUnit[44] := "gs";
asLeakTesterUnit[45] := "gm";
asLeakTesterUnit[46] := "degC";
asLeakTesterUnit[47] := "degF";
asLeakTesterUnit[48] := "degK";
asLeakTesterUnit[49] := "hour";
asLeakTesterUnit[50] := "min";
asLeakTesterUnit[51] := "sec";
asLeakTesterUnit[52] := "msec";
asLeakTesterUnit[53] := "yr";
asLeakTesterUnit[54] := "mth";
asLeakTesterUnit[55] := "wk";
asLeakTesterUnit[56] := "day";
asLeakTesterUnit[57] := "cc";
asLeakTesterUnit[58] := "cin";
asLeakTesterUnit[59] := "l";
asLeakTesterUnit[60] := "gal";
asLeakTesterUnit[61] := "mL";
asLeakTesterUnit[62] := "in";
asLeakTesterUnit[63] := "mic";
asLeakTesterUnit[64] := "cm";
asLeakTesterUnit[65] := "mm";
asLeakTesterUnit[66] := "M";
asLeakTesterUnit[67] := "thou";
asLeakTesterUnit[68] := "mil";
asLeakTesterUnit[69] := "V";
asLeakTesterUnit[70] := "mV";
asLeakTesterUnit[71] := "uV";
asLeakTesterUnit[72] := "A";
asLeakTesterUnit[73] := "mA";
asLeakTesterUnit[74] := "uA";
asLeakTesterUnit[75] := "dB";
asLeakTesterUnit[76] := "bits";
asLeakTesterUnit[77] := "ppm";
asLeakTesterUnit[78] := "PF";
asLeakTesterUnit[79] := "%";
asLeakTesterUnit[80] := "unit";
asLeakTesterUnit[81] := "cnts";
asLeakTesterUnit[82] := "atm/s";
asLeakTesterUnit[83] := "bar/s";
asLeakTesterUnit[84] := "cHg/s";
asLeakTesterUnit[85] := "inHg/s";
asLeakTesterUnit[86] := "kPa/s";
asLeakTesterUnit[87] := "psi/s";
asLeakTesterUnit[88] := "iWC/s";
asLeakTesterUnit[89] := "cWC/s";
asLeakTesterUnit[90] := "mWC/s";
asLeakTesterUnit[91] := "ksc/s";
asLeakTesterUnit[92] := "g/a";
asLeakTesterUnit[93] := "oz/yr";
asLeakTesterUnit[94] := "ppm";
asLeakTesterUnit[95] := "mbl/s";
asLeakTesterUnit[96] := "Pam/s";
asLeakTesterUnit[97] := "acc/s";
asLeakTesterUnit[98] := "Trl/s";
asLeakTesterUnit[99] := "Pam/h";
asLeakTesterUnit[100] := "gr/yr";
asLeakTesterUnit[101] := "lb/yr";
asLeakTesterUnit[102] := "acc/m";
asLeakTesterUnit[103] := "kg";
asLeakTesterUnit[104] := "g";
asLeakTesterUnit[105] := "lb";
asLeakTesterUnit[106] := "oz";
asLeakTesterUnit[107] := "MPa/s";
asLeakTesterUnit[108] := "mb/s";
asLeakTesterUnit[109] := "mHg/s";
asLeakTesterUnit[110] := "pa/s";
asLeakTesterUnit[111] := "MPa/s";
END_ACTION

ACTION ACT_LiveSegmentCode:
asLeakTesterSegments[0] := "NO DATA";
asLeakTesterSegments[1] := "INTERN PreSeq";
asLeakTesterSegments[2] := "Intern PostSeq";
asLeakTesterSegments[3] := "Intern EmptySeq";
asLeakTesterSegments[4] := "Intern - Evaluate Part Result";
asLeakTesterSegments[5] := "Setup - Pre-Seq";
asLeakTesterSegments[6] := "Setup - Post-Seq";
asLeakTesterSegments[7] := "Setup - Pressure Select";
asLeakTesterSegments[8] := "Setup - Manifold Fill";
asLeakTesterSegments[9] := "Setup - Manifold Isolate";
asLeakTesterSegments[10] := "Setup - Manifold Exhaust";
asLeakTesterSegments[11] := "Prefill til Pressure";
asLeakTesterSegments[12] := "Prefill";
asLeakTesterSegments[13] := "Prefill Pre-Pressure";
asLeakTesterSegments[14] := "Prefill - Charge Volume";
asLeakTesterSegments[15] := "Fill References";
asLeakTesterSegments[16] := "Fill (without pressure monitoring)";
asLeakTesterSegments[17] := "Fill Ramp";
asLeakTesterSegments[18] := "Fill Tracer";
asLeakTesterSegments[19] := "Fill Tracer Gross";
asLeakTesterSegments[20] := "Fill Step";
asLeakTesterSegments[21] := "Fill Evac";
asLeakTesterSegments[22] := "Fill Clean";
asLeakTesterSegments[23] := "Fill til Full";
asLeakTesterSegments[24] := "Stabilize Tracer";
asLeakTesterSegments[25] := "Stabilize Tracer Gross";
asLeakTesterSegments[26] := "Stabilize DP Xder Balance";
asLeakTesterSegments[27] := "Stabilize Evac";
asLeakTesterSegments[28] := "Stabilize Step Dwell";
asLeakTesterSegments[29] := "Stabilize Chamber Cleanup";
asLeakTesterSegments[30] := "Stabilize til Slope";
asLeakTesterSegments[31] := "Stabilize DP";
asLeakTesterSegments[32] := "Stabilize Xder Test";
asLeakTesterSegments[33] := "Stabilize Flow";
asLeakTesterSegments[34] := "Stabilize References Volume";
asLeakTesterSegments[35] := "Stabilize Tracer Wait";
asLeakTesterSegments[36] := "Stabilize Balance DP";
asLeakTesterSegments[37] := "Pressure Decay - Leak Standard Test";
asLeakTesterSegments[38] := "Rate Pressure Loss Test";
asLeakTesterSegments[39] := "Occlusion Test (Backpressure)";
asLeakTesterSegments[40] := "Percent References Volume Test";
asLeakTesterSegments[41] := "Pressure Loss Test";
asLeakTesterSegments[42] := "Ramp Pressure Event Test";
asLeakTesterSegments[43] := "Proof Test";
asLeakTesterSegments[44] := "Ramp Flow Event Test";
asLeakTesterSegments[45] := "Refrigerant Fill";
asLeakTesterSegments[46] := "Ramp Digital Input Event Test";
asLeakTesterSegments[47] := "Sniffer Test";
asLeakTesterSegments[48] := "Sniffer Gross Test";
asLeakTesterSegments[49] := "Step Proof";
asLeakTesterSegments[50] := "Differential Pressure Decay - Leak Standard Test";
asLeakTesterSegments[51] := "Evac Test";
asLeakTesterSegments[52] := "Differential Pressure Decay Test";
asLeakTesterSegments[53] := "Differential Pressure Decay Test (no absl pressure)";
asLeakTesterSegments[54] := "Precise Mass Flow Test (Differential Flow)";
asLeakTesterSegments[55] := "Mass Flow Test";
asLeakTesterSegments[56] := "Mass Flow - Leak Rate Test";
asLeakTesterSegments[57] := "Differential Pressure Decay - Leak Standard Test (no absl pressure)";
asLeakTesterSegments[58] := "Differential Pressure Decay - Leak Rate (volume calculated)";
asLeakTesterSegments[59] := "Pressure Switch Test";
asLeakTesterSegments[60] := "Transducer Test";
asLeakTesterSegments[61] := "Pressure Verify";
asLeakTesterSegments[62] := "Exhaust";
asLeakTesterSegments[63] := "Exhaust til Pressure";
asLeakTesterSegments[64] := "Exhaust til Input";
asLeakTesterSegments[65] := "Exhaust til Analog Input";
asLeakTesterSegments[66] := "Exhaust til Slope";
asLeakTesterSegments[67] := "Exhaust til Empty";
asLeakTesterSegments[68] := "Exhaust - Re-Evacuate";
asLeakTesterSegments[69] := "Exhaust - T-Gas";
asLeakTesterSegments[70] := "Exhaust - Chamber Output Rest";
asLeakTesterSegments[71] := "Verify Pressure";
asLeakTesterSegments[72] := "Verify Pressure after Delay";
asLeakTesterSegments[73] := "Verify Input";
asLeakTesterSegments[74] := "Verify Input after Delay";
asLeakTesterSegments[75] := "Verify Analog Input";
asLeakTesterSegments[76] := "Verify Analog Input after Delay";
asLeakTesterSegments[77] := "Verify Slope";
asLeakTesterSegments[78] := "Verify Slope after Delay";
asLeakTesterSegments[79] := "Drive Output";
asLeakTesterSegments[80] := "Drive Output Period";
asLeakTesterSegments[81] := "Drive Analog Output";
asLeakTesterSegments[82] := "Drive Analog Output Period";
asLeakTesterSegments[83] := "Drive Valve";
asLeakTesterSegments[84] := "Drive Valve Period";
asLeakTesterSegments[85] := "Link Control";
asLeakTesterSegments[86] := "Link Decision";
asLeakTesterSegments[87] := "Autorun Relax";
asLeakTesterSegments[88] := "Calibration Relax";
asLeakTesterSegments[89] := "Delay";
asLeakTesterSegments[90] := "Pressure Transducer Zero";
asLeakTesterSegments[91] := "Flow Transducer Zero";
asLeakTesterSegments[92] := "Differential Pressure Transducer Zero";
asLeakTesterSegments[93] := "Pressure Select (Range Only)";
asLeakTesterSegments[94] := "Pressure Select (Evac)";
asLeakTesterSegments[95] := "Pressure Select";
asLeakTesterSegments[96] := "Pressure Select (Ramp)";
asLeakTesterSegments[97] := "Pressure Select (Tracer)";
asLeakTesterSegments[98] := "Pressure Select (Clean)";
asLeakTesterSegments[99] := "Pressure Select (None)";
asLeakTesterSegments[100] := "Tooling Motion Control";
asLeakTesterSegments[101] := "Tooling Motion Extend";
asLeakTesterSegments[102] := "Tooling Motion Retract";
asLeakTesterSegments[103] := "Tooling Part Mark";
asLeakTesterSegments[104] := "Tooling Seal Extend";
asLeakTesterSegments[105] := "Tooling Seal Retract";
asLeakTesterSegments[106] := "External Volume";
asLeakTesterSegments[107] := "Setup - Set Regulator";
asLeakTesterSegments[108] := "Setup - Electronic Regulator Analyze";
asLeakTesterSegments[109] := "Setup - Electronic Regulator Zero";
asLeakTesterSegments[110] := "Setup - Electronic Regulator Setpoint";
asLeakTesterSegments[111] := "Setup - Transducer Residual";
asLeakTesterSegments[112] := "Setup - Pressure Transducer Zero";
asLeakTesterSegments[113] := "Setup - Flow Transducer Zero";
asLeakTesterSegments[114] := "Setup - Pressure Transducer Setpoint";
asLeakTesterSegments[115] := "Setup - Flow Transducer Setpoint";
asLeakTesterSegments[116] := "Setup - DP Transducer Setpoint";
asLeakTesterSegments[117] := "Setup - Pressure Transducer Verification";
asLeakTesterSegments[118] := "Setup - Flow Transducer Verification";
asLeakTesterSegments[119] := "Setup - Sniffer Init 1";
asLeakTesterSegments[120] := "Setup - Sniffer Init 2";
asLeakTesterSegments[121] := "Setup - Sniffer Idle";
asLeakTesterSegments[122] := "Setup - Mix Verification";
asLeakTesterSegments[123] := "Setup - Scale Init";
asLeakTesterSegments[124] := "Setup - Atmospheric Pressure Check";
asLeakTesterSegments[125] := "Setup - DP Transducer Zero";
asLeakTesterSegments[126] := "Setup - DP Transducer Verification";
asLeakTesterSegments[127] := "Begin Chamber Functions";
asLeakTesterSegments[128] := "Chamber - hardvac control";
asLeakTesterSegments[129] := "Chamber - blower control";
asLeakTesterSegments[130] := "Chamber - inlet blower on";
asLeakTesterSegments[131] := "Chamber - inlet blower off";
asLeakTesterSegments[132] := "Chamber - circulation on";
asLeakTesterSegments[133] := "Chamber - outlet blower on";
asLeakTesterSegments[134] := "Chamber - outlet blower off";
asLeakTesterSegments[135] := "Chamber - circulation off";
asLeakTesterSegments[136] := "Chamber - accumulation rest";
asLeakTesterSegments[137] := "Chamber - clamshell purge rings control";
asLeakTesterSegments[138] := "Chamber - clamshell purge rings option";
asLeakTesterSegments[139] := "Chamber - clamshell purge rings rest";
asLeakTesterSegments[140] := "Chamber - Exh";
asLeakTesterSegments[141] := "Chamber - vent off";
asLeakTesterSegments[142] := "Chamber - evacuate on";
asLeakTesterSegments[143] := "Chamber - evacuate off";
asLeakTesterSegments[144] := "Chamber - pre-purge";
asLeakTesterSegments[145] := "Refrigerant CS Isolation";
asLeakTesterSegments[146] := "Refrigerant Stabilize";
asLeakTesterSegments[147] := "Refrigerant Part Switch";
asLeakTesterSegments[148] := "Refrigerant Vent";
asLeakTesterSegments[149] := "Refrigerant Iso Off";
asLeakTesterSegments[150] := "Stabilize Scale";
asLeakTesterSegments[151] := "Refrigerant Manual Fill";
asLeakTesterSegments[152] := "Refrigerant Evac";
END_ACTION

ACTION ACT_Precision:
asLeakTesterPrecision[0] := "NO DATA";
asLeakTesterPrecision[1] := "Digits of precision: X";
asLeakTesterPrecision[2] := "Digits of precision: X.X";
asLeakTesterPrecision[3] := "Digits of precision: X.XX";
asLeakTesterPrecision[4] := "Digits of precision: X.XXX";
asLeakTesterPrecision[5] := "Digits of precision: X.XXXX";
asLeakTesterPrecision[6] := "Digits of precision: X.XXXXX";
END_ACTION

ACTION ACT_ProgramEvaluation:
asLeakTesterProgramEvaluation[0] := "NO DATA";
asLeakTesterProgramEvaluation[1] := "TEST PASSED";
asLeakTesterProgramEvaluation[2] := "TEST FAILED";
asLeakTesterProgramEvaluation[3] := "TEST ERROR";
asLeakTesterProgramEvaluation[4] := "TEST SKIPPED";
asLeakTesterProgramEvaluation[5] := "TEST FAILED - LEVEL 1";
asLeakTesterProgramEvaluation[6] := "TEST FAILED - LEVEL 2";
asLeakTesterProgramEvaluation[7] := "TEST FAILED - LEVEL 3";
asLeakTesterProgramEvaluation[8] := "AUTO-CAL MASTER PART";
asLeakTesterProgramEvaluation[9] := "AUTO-CAL LEAK STANDARD PART";
asLeakTesterProgramEvaluation[10] := "TEST FAILED - NO EVENT";
asLeakTesterProgramEvaluation[11] := "TEST COMPLETE";
END_ACTION

ACTION ACT_TestType:
asLeakTesterTestType[0] := "NO DATA";
asLeakTesterTestType[1] := "Pressure Decay - Leak Standard Test";
asLeakTesterTestType[2] := "Rate of Pressure Loss Test";
asLeakTesterTestType[3] := "Occlusion Test (Backpressure)";
asLeakTesterTestType[4] := "Percent of Reference Volume Tes";
asLeakTesterTestType[5] := "Pressure Loss Test";
asLeakTesterTestType[6] := "Ramp to Pressure Event Test";
asLeakTesterTestType[7] := "Proof Test";
asLeakTesterTestType[8] := "Ramp to Flow Event Test";
asLeakTesterTestType[9] := "Refrigerant Fill";
asLeakTesterTestType[10] := "Ramp to Digital Input Event Test";
asLeakTesterTestType[11] := "Sniffer Test";
asLeakTesterTestType[12] := "";
asLeakTesterTestType[13] := "Sniffer Gross Test";
asLeakTesterTestType[14] := "Step Proof";
asLeakTesterTestType[15] := "Differential Pressure Decay - Leak | Standard Test";
asLeakTesterTestType[16] := "Evac Test";
asLeakTesterTestType[17] := "Differential Pressure Decay Test";
asLeakTesterTestType[18] := "Differential Pressure Decay Test (no abs pressure)";
asLeakTesterTestType[19] := "Precise Mass Flow Test (Differential Flow)";
asLeakTesterTestType[20] := "Mass Flow Test";
asLeakTesterTestType[21] := "Mass Flow - Leak Rate Test";
asLeakTesterTestType[22] := "Differential Pressure Decay - Leak Standard Test (no abs pressure)";
asLeakTesterTestType[23] := "Differential Pressure Decay - Leak Rate (volume calculated)";
asLeakTesterTestType[24] := "Pressure Switch Test";
asLeakTesterTestType[25] := "Transducer Test";
END_ACTION

END_PROGRAM

// ---- POUs/G_Utility/FB_Alarms.TcPOU
FUNCTION_BLOCK FB_Alarms
VAR_INPUT
	evEntry			: TcEventEntry;
	bEvt			: BOOL;
	bConfirm		: BOOL;
END_VAR
VAR_OUTPUT
	Q							: BOOL;
END_VAR
VAR
	bInit			: BOOL :=	TRUE;
	rAlarmActivation: Tc2_Standard.R_TRIG;
	rReset			: Tc2_Standard.RS;
END_VAR

IF bInit THEN
	
	SUPER^.CreateEx(evEntry, TRUE, 0);
	bInit := FALSE;

END_IF


IF bEvt  THEN
	SUPER^.Raise (0);
ELSE SUPER^.Clear (0, FALSE);
END_IF


IF bConfirm AND NOT bEvt THEN
	
	SUPER^.Confirm(0);

END_IF


Q := SUPER^.bRaised;

END_FUNCTION_BLOCK

// ---- POUs/G_Utility/FB_BoxInfo.TcPOU
FUNCTION_BLOCK FB_BoxInfo
VAR_INPUT
	  nPnIoBoxState : UINT;    	
      nPnIoBoxDiag  : UINT;
END_VAR
VAR_OUTPUT
		sBoxState     : STRING;
	  sBoxDiag      : STRING;
END_VAR
VAR
END_VAR


IF nPnIoBoxState = 0 THEN 
	sBoxState := 'No error';
ELSIF nPnIoBoxState = 1 THEN 
	sBoxState := 'Profinet device state machine is in boot mode';
ELSIF nPnIoBoxState = 2 THEN 
	sBoxState := 'Device not found';
ELSIF nPnIoBoxState = 3 THEN 
	sBoxState := 'The stationname is not unique';
ELSIF nPnIoBoxState = 4 THEN 
	sBoxState := 'IP could not be set';
ELSIF nPnIoBoxState = 5 THEN 
	sBoxState := 'IP conflict';
ELSIF nPnIoBoxState = 6 THEN 
	sBoxState := 'DCP set was not successful';
ELSIF nPnIoBoxState = 7 THEN 
	sBoxState := 'Watchdog error';
ELSIF nPnIoBoxState = 8 THEN 
	sBoxState := 'Datahold error';
ELSIF nPnIoBoxState = 9 THEN 
	sBoxState := 'RTC3: Sync mode could not be initiated';
ELSIF nPnIoBoxState = 10 THEN 
	sBoxState := 'Profinet controller has a link error';
ELSIF nPnIoBoxState = 11 THEN 
	sBoxState := 'The aliasname is not unique';
ELSIF nPnIoBoxState = 12 THEN 
	sBoxState := 'The automatic name assignement isnt possible - wrong device type';	
ELSIF nPnIoBoxState = 13 THEN 
	sBoxState := 'IOC-AR is established but no application ready';	
ELSIF nPnIoBoxState = 14 THEN 
	sBoxState := 'IOC-AR is established but module difference';	
ELSIF nPnIoBoxState = 15 THEN 
	sBoxState := 'At least one InputCR is invalid, provider in stop or problemindicator is set';
ELSIF nPnIoBoxState = 16 THEN 
	sBoxState := 'At least one OutputCR is invalid, provider in stop or problemindicator is set';
ELSIF nPnIoBoxState = 31 THEN 
	sBoxState := 'Only for EtherCAT gateways: WC-State of cyclic EtherCAT frame is 1';	
END_IF

IF nPnIoBoxDiag = 0 THEN
   sBoxDiag := 'No diagnosis';
ELSIF nPnIoBoxDiag = 16#0001 THEN
   sBoxDiag := 'IOC-AR is not established'; 
ELSIF nPnIoBoxDiag = 16#0002 THEN
   sBoxDiag := 'IOC-AR is established'; 
ELSIF nPnIoBoxDiag = 16#0004 THEN
   sBoxDiag := 'IOC-AR is established but no application ready'; 
ELSIF nPnIoBoxDiag = 16#0008 THEN
   sBoxDiag := 'IOC-AR is established but module difference'; 
ELSIF nPnIoBoxDiag = 16#0010 THEN
   sBoxDiag := 'At least one AlarmCR got a diagnosis alarm'; 
ELSIF nPnIoBoxDiag = 16#0100 THEN
   sBoxDiag := 'At least one InputCR is invalid'; 
ELSIF nPnIoBoxDiag = 16#0200 THEN
   sBoxDiag := 'At least one InputCR Provider is in stop'; 
ELSIF nPnIoBoxDiag = 16#0400 THEN
   sBoxDiag := 'At least one InputCR Problemindicator is set';    
ELSIF nPnIoBoxDiag = 16#1000 THEN
   sBoxDiag := 'At least one OutputCR is invalid';    
ELSIF nPnIoBoxDiag = 16#2000 THEN
   sBoxDiag := 'At least one OutputCR Provider is in stop';    
ELSIF nPnIoBoxDiag = 16#4000 THEN
   sBoxDiag := 'At least one OutputCR Problemindicator is set';    
END_IF

END_FUNCTION_BLOCK

// ---- POUs/G_Utility/FB_DayOfYear.TcPOU
FUNCTION_BLOCK FB_DayOfYear
VAR_INPUT
	nMonth : UINT;
	nDay : UINT;
END_VAR
VAR_OUTPUT
	nDayOfYear : UINT;
END_VAR
VAR
	nDayTemp : UINT;
END_VAR

IF nMonth =1 THEN
	nDayTemp := 0;
ELSIF nMonth =2 THEN
	nDayTemp := 31;
ELSIF nMonth =3 THEN
	nDayTemp := 59;
ELSIF nMonth =4 THEN
	nDayTemp := 90;
ELSIF nMonth =5 THEN
	nDayTemp := 120;	
ELSIF nMonth =6 THEN
	nDayTemp := 151;
ELSIF nMonth =7 THEN
	nDayTemp := 161;
ELSIF nMonth =8 THEN
	nDayTemp := 212;
ELSIF nMonth =9 THEN
	nDayTemp := 243;
ELSIF nMonth =10 THEN
	nDayTemp := 273;
ELSIF nMonth =11 THEN
	nDayTemp := 304;
ELSIF nMonth =12 THEN
	nDayTemp := 334;	
END_IF
nDayOFYear := nDayTemp + nDay;

END_FUNCTION_BLOCK

// ---- POUs/G_Utility/FB_HeightMeasurement.TcPOU
FUNCTION_BLOCK FB_HeightMeasurement
VAR_INPUT

	aSensorCurrentValue							: ARRAY[1..4] OF DINT;
	bEnable										: BOOL;
	bMeasurementRequest							: BOOL;
	
	
	bSet										: BOOL;
	aTolerance									: ARRAY[1..4] OF DINT;

	
	bManualMode									: BOOL;
	bManualMeasure								: BOOL;
	bAcknowledge								: BOOL;
	bFunctionFault								: BOOL;
	
	
	
	
END_VAR
VAR_OUTPUT
	bBusy										: BOOL;
	bComplete									: BOOL;
	bEnableo									: BOOL;
	wFunctionState								: STRING;
	nSensorSetPoint								: ARRAY[1..4] OF DINT;
	aPass										: ARRAY[1..5] OF BOOL; //5 Final Result
	aFail										: ARRAY[1..5] OF BOOL; //5 Final Result
	aMinLimit									: ARRAY[1..4] OF DINT;
	aMaxLimit									: ARRAY[1..4] OF DINT;

	
END_VAR
VAR
	i											: INT;
	j											: INT;
	nFunctionProcess							: INT;
	nReference									: DINT;
	
	tonCaseDelay								: ARRAY[0..10] OF TON;
	rtrigCaseTriger								: ARRAY[0..10] OF R_TRIG;
END_VAR

ACT_TimTrig();

IF NOT bEnable THEN
	nFunctionProcess			:= 0;
	bEnableo					:= FALSE;
ELSE 
	bEnableo					:= TRUE;
END_IF





CASE nFunctionProcess OF 

0:
wFunctionState				:='Function Disabled';
bBusy						:= FALSE;
IF bEnable THEN
	nFunctionProcess		:=1;
END_IF

1:
wFunctionState				:='Waiting';
IF tonCaseDelay[5].Q THEN
	nFunctionProcess		:=2;
END_IF
2:
j							:= 0;
ACT_Fault();
IF bFunctionFault THEN
	nFunctionProcess		:=50;
ELSIF bMeasurementRequest THEN
	nFunctionProcess		:=10;
ELSIF	bManualMode THEN
	nFunctionProcess		:=30;
END_IF

10:
j							:= 0;
FOR j:=1 TO 5 DO
	
	aPass[j] 				:= FALSE;
	aFail[j] 				:= FALSE;
	
END_FOR
IF tonCaseDelay[6].Q THEN
	nFunctionProcess		:=11;
END_IF
11:
wFunctionState				:='Working';
bBusy						:= TRUE;
IF tonCaseDelay[0].Q THEN
	nFunctionProcess		:=13;
END_IF

13:
FOR j:=1 TO 4 DO
	IF aSensorCurrentValue[j] < aMaxLimit[j] AND  aSensorCurrentValue[j] > aMinLimit[j] THEN
		aPass[j] := TRUE;
	ELSE aFail[j] := TRUE;
	END_IF
END_FOR
IF tonCaseDelay[1].Q THEN
	nFunctionProcess		:=14;
	j						:= 0;
END_IF

14:
aPass[5]					:= TRUE;
aFail[5]					:= FALSE;
FOR j:=1 TO 4 DO
IF aFail[j] THEN
	aPass[5]				:= FALSE;
	aFail[5]				:= TRUE;
END_IF
END_FOR
IF tonCaseDelay[3].Q THEN
	nFunctionProcess		:=16;
END_IF

16:
wFunctionState				:='Process Complete';
bComplete					:= TRUE;
bBusy						:= FALSE;
j							:= 0;
IF bAcknowledge  THEN	
	nFunctionProcess		:=20;
END_IF

20:
bComplete	:= FALSE;
IF tonCaseDelay[2].Q THEN
	nFunctionProcess		:=1;
END_IF

30:
wFunctionState				:='Manual Mode';
IF bManualMode THEN
	ACT_Manual();
ELSIF bFunctionFault THEN
	nFunctionProcess		:=50;
ELSE nFunctionProcess		:=1;
END_IF




50: 
wFunctionState				:='Error';
IF tonCaseDelay[4].Q THEN
	nFunctionProcess		:=1;
END_IF



END_CASE

ACTION ACT_Fault:
(*FOR i:=1 TO 5 DO
	IF aCurrentValueInvalid[i] OR aCurrentValueUnderRange[i] OR aCurrentValueOverRange[i] OR aSensorErrorStatus[i] OR bTerminalErrorStatus THEN 

	bFunctionFault := TRUE;
	
	ELSE bFunctionFault := FALSE;
	
	END_IF

END_FOR
IF GVL_MASTER.bFlash1Hz THEN
	i:=0;
END_IF*)
END_ACTION

ACTION ACT_Manual:
	

	aMinLimit[1]		:= nSensorSetPoint[1] - aTolerance[1];
	aMinLimit[2]		:= nSensorSetPoint[2] - aTolerance[2];
	aMinLimit[3]		:= nSensorSetPoint[3] - aTolerance[3];
	aMinLimit[4]		:= nSensorSetPoint[4] - aTolerance[4];
	
	aMaxLimit[1]		:= nSensorSetPoint[1] + aTolerance[1];
	aMaxLimit[2]		:= nSensorSetPoint[2] + aTolerance[2];
	aMaxLimit[3]		:= nSensorSetPoint[3] + aTolerance[3];
	aMaxLimit[4]		:= nSensorSetPoint[4] + aTolerance[4];

IF bSet THEN
	
	nSensorSetPoint[1] 	:= aSensorCurrentValue[1];
	nSensorSetPoint[2] 	:= aSensorCurrentValue[2];
	nSensorSetPoint[3] 	:= aSensorCurrentValue[3];
	nSensorSetPoint[4] 	:= aSensorCurrentValue[4];
	

	
END_IF

IF bManualMeasure THEN
	aPass[5]					:= TRUE;
	aFail[5]					:= FALSE;
	FOR j:=1 TO 4 DO
		IF aSensorCurrentValue[j] <= aMaxLimit[j] AND  aSensorCurrentValue[j] >= aMinLimit[j] THEN
			aPass[j] := TRUE;
			aFail[j] := FALSE;
		ELSE 
			aFail[j] := TRUE;
			aPass[j] := FALSE;
			
		END_IF
		IF aFail[j] THEN
		aPass[5]				:= FALSE;
		aFail[5]				:= TRUE;
		END_IF
	END_FOR
	

	
END_IF
END_ACTION

ACTION ACT_TimTrig:
tonCaseDelay[0](IN:= nFunctionProcess = 11,PT:=T#3S);
tonCaseDelay[1](IN:= nFunctionProcess = 13,PT:=T#1S);
tonCaseDelay[2](IN:= nFunctionProcess = 20,PT:=T#1S);
tonCaseDelay[3](IN:= nFunctionProcess = 14,PT:=T#1S);
tonCaseDelay[4](IN:= nFunctionProcess = 50 AND NOT bFunctionFault,PT:=T#1S);
tonCaseDelay[5](IN:= nFunctionProcess = 1,PT:=T#1S);
tonCaseDelay[6](IN:=nFunctionProcess = 10 ,PT:=T#1S);
tonCaseDelay[7](IN:= ,PT:=T#2S);

//rtrigCaseTriger[0]();
END_ACTION

END_FUNCTION_BLOCK

// ---- POUs/G_Utility/FB_HeightTest.TcPOU
FUNCTION_BLOCK FB_HeightTest
VAR_INPUT
	
	
	bEnableFunct   : BOOL;
	bStartMesure   : BOOL;
	bPuls          : BOOL;
	bAknwResult    : BOOL;
	bReference     : ARRAY[1..4] OF BOOL;
	nRawMesure     : ARRAY[1..4] OF DINT;
	rSetPoint      : ARRAY[1..4] OF REAL;
    rTolerance     : ARRAY[1..4] OF REAL;


END_VAR
VAR_OUTPUT
	
	rMesureDis     : ARRAY[1..4] OF REAL; // 
    rMesuredValue  : ARRAY[1..4] OF REAL; // Converted mesure to value Real
	bMesOutOfToler : ARRAY[1..4] OF BOOL; // Mesure out of Tolerance
	bMesFuncFault  : BOOL; // Parametore of Inspection not choose
	bSetPointFault : BOOL;
	bTolerFault    : BOOL;
	bWaitToAknw    : BOOL;
	bBusyMesure    : BOOL;
	
END_VAR

VAR_IN_OUT
    stMesureStat   : ARRAY[0..4] OF ST_MeasureStatistics;
END_VAR

VAR
	rRawMesureConv : ARRAY[1..4] OF REAL;
    nMesureFunc    : UINT;
	rTolerTempCal  : ARRAY[1..4] OF REAL;
	nMesureSeq     : INT :=10;
	nTempSeqStep   : INT;
	tonSequTim     : ARRAY[1..20] OF Tc2_Standard.TON;
	rtrigSeqTrig   : ARRAY[1..20] OF Tc2_Standard.R_TRIG;
	bSetpChanged   : BOOL;
END_VAR

// Conv to mikro m 
rRawMesureConv[1] := (DINT_TO_REAL(nRawMesure[1]))/10.0;
rMesuredValue[1]  := rRawMesureConv[1];

rRawMesureConv[2] := (DINT_TO_REAL(nRawMesure[2]))/10.0;
rMesuredValue[2]  := rRawMesureConv[2];

rRawMesureConv[3] := (DINT_TO_REAL(nRawMesure[3]))/10.0;
rMesuredValue[3]  := rRawMesureConv[3];

rRawMesureConv[4] := (DINT_TO_REAL(nRawMesure[4]))/10.0;
rMesuredValue[4]  := rRawMesureConv[4]; 

IF bEnableFunct AND bReference[1] THEN
   nMesureFunc := 1;
ELSIF bEnableFunct AND bReference[2] THEN
   nMesureFunc := 2; 
ELSIF bEnableFunct AND bReference[3] THEN
   nMesureFunc := 3;
ELSIF bEnableFunct AND bReference[4] THEN
   nMesureFunc := 4;
ELSE
   nMesureFunc := 5;  
END_IF

bWaitToAknw := (nMesureSeq=150) OR (nMesureSeq=250) OR (nMesureSeq=350) OR (nMesureSeq=450);

bSetPointFault:= (rSetPoint[1] = 0) OR (rSetPoint[2] = 0) OR (rSetPoint[3] = 0) OR (rSetPoint[4] = 0);
bTolerFault:= (rTolerance[1] = 0) OR (rTolerance[1] = 0) OR (rTolerance[3] = 0) OR (rTolerance[4] = 0);
// Timers and Triggers
tonSequTim[1](IN:=(nMesureSeq=500) ,PT:= T#100MS);
tonSequTim[2](IN:=(nMesureSeq=150) ,PT:= T#200MS);
tonSequTim[3](IN:=(nMesureSeq=250) ,PT:= T#200MS);
tonSequTim[4](IN:=(nMesureSeq=350) ,PT:= T#200MS);
tonSequTim[5](IN:=(nMesureSeq=450) ,PT:= T#200MS);
rtrigSeqTrig[1](CLK:= (bPuls));
rtrigSeqTrig[2](CLK:=bAknwResult);
rtrigSeqTrig[3](CLK:=(NOT bEnableFunct));
//---------------------------
bSetpChanged:= rtrigSeqTrig[1].Q;
 
IF rtrigSeqTrig[3].Q THEN
	bMesOutOfToler[1]:= FALSE;
    bMesOutOfToler[2]:= FALSE;
	bMesOutOfToler[3]:= FALSE;
	bMesOutOfToler[4]:= FALSE;
	nMesureSeq := 10;
END_IF

bBusyMesure:= bEnableFunct  AND nMesureSeq>10 AND nMesureSeq<500;
CASE  nMesureSeq OF
10:
   IF nMesureFunc = 1 AND bStartMesure THEN
	nTempSeqStep:= 10;
	nMesureSeq := 100;
ELSIF nMesureFunc = 2 AND bStartMesure THEN
	nTempSeqStep:= 10;
	nMesureSeq := 200;
ELSIF nMesureFunc = 3 AND bStartMesure THEN
	nTempSeqStep:= 10;
	nMesureSeq := 300;
ELSIF nMesureFunc = 4 AND bStartMesure THEN
	nTempSeqStep:= 10;
	nMesureSeq := 400;
ELSIF nMesureFunc = 5 AND bStartMesure THEN
	nTempSeqStep:= 10;
	nMesureSeq := 500; 	
END_IF
    stMesureStat[1].bOutLimitMin := FALSE;
    stMesureStat[1].bOutLimitMax := FALSE;	
    stMesureStat[2].bOutLimitMin := FALSE;
    stMesureStat[2].bOutLimitMax := FALSE;	
    stMesureStat[3].bOutLimitMin := FALSE;
    stMesureStat[3].bOutLimitMax := FALSE;	
    stMesureStat[4].bOutLimitMin := FALSE;
    stMesureStat[4].bOutLimitMax := FALSE; 
//=========================================================================================================
100: // Variable 1 choose for reference point
rMesureDis[1] := rSetPoint[1] - rMesuredValue[1]; // Diference  on Distance mesure 1
IF bSetpChanged THEN
	nTempSeqStep:= 100;
	nMesureSeq := 105; 
END_IF
105:// If it is in Tolerance
IF rMesureDis[1]<rSetPoint[1]-rTolerance[1] OR rMesureDis[1]>rSetPoint[1]+rTolerance[1] THEN
bMesOutOfToler[1]:= TRUE;
ELSE
bMesOutOfToler[1]:= FALSE;	
END_IF
// Statistic
IF rMesureDis[1]<rSetPoint[1]-rTolerance[1] THEN
	stMesureStat[1].bOutLimitMin := TRUE;
ELSIF rMesureDis[1]>rSetPoint[1]+rTolerance[1] THEN
	stMesureStat[1].bOutLimitMax := TRUE;
ELSE
    stMesureStat[1].bOutLimitMin := FALSE;
    stMesureStat[1].bOutLimitMax := FALSE; 	
END_IF

IF bSetpChanged THEN
	nTempSeqStep:= 105;
	nMesureSeq := 110; 
END_IF
110:// Mesure 2 value 
rMesureDis[2]:= rMesuredValue[2] - rMesuredValue[1];
IF bSetpChanged THEN
	nTempSeqStep:= 110;
	nMesureSeq := 115; 
END_IF
115:// If it is in Tolerance
IF rMesureDis[2]<rSetPoint[2]-rTolerance[2] OR rMesureDis[2]>rSetPoint[2]+rTolerance[2] THEN
bMesOutOfToler[2]:= TRUE;
ELSE
bMesOutOfToler[2]:= FALSE;	
END_IF
// Statistic ========================================
IF rMesureDis[2]<rSetPoint[2]-rTolerance[2] THEN
	stMesureStat[2].bOutLimitMin := TRUE;
ELSIF rMesureDis[2]>rSetPoint[2]+rTolerance[2] THEN
	stMesureStat[2].bOutLimitMax := TRUE;
ELSE
    stMesureStat[2].bOutLimitMin := FALSE;
    stMesureStat[2].bOutLimitMax := FALSE; 	
END_IF
//===================================================
IF bSetpChanged THEN
	nTempSeqStep:= 115;
	nMesureSeq := 120; 
END_IF
120: // Mesure 3 value 
rMesureDis[3]:= rMesuredValue[3] - rMesuredValue[1];
IF bSetpChanged THEN
	nTempSeqStep:= 120;
	nMesureSeq := 125; 
END_IF
125:// If it is in Tolerance
IF rMesureDis[3]<rSetPoint[3]-rTolerance[3] OR rMesureDis[3]>rSetPoint[3]+rTolerance[3] THEN
bMesOutOfToler[3]:= TRUE;
ELSE
bMesOutOfToler[3]:= FALSE;	
END_IF
// Statistic ========================================
IF rMesureDis[3]<rSetPoint[3]-rTolerance[3] THEN
	stMesureStat[3].bOutLimitMin := TRUE;
ELSIF rMesureDis[3]>rSetPoint[3]+rTolerance[3] THEN
	stMesureStat[3].bOutLimitMax := TRUE;
ELSE
    stMesureStat[3].bOutLimitMin := FALSE;
    stMesureStat[3].bOutLimitMax := FALSE; 	
END_IF
//===================================================
IF bSetpChanged THEN
	nTempSeqStep:= 125;
	nMesureSeq := 140; 
END_IF
140:  // Mesure 4 value 
rMesureDis[4]:= rMesuredValue[4] - rMesuredValue[1];
IF bSetpChanged THEN
	nTempSeqStep:= 140;
	nMesureSeq := 145; 
END_IF
145:// If it is in Tolerance
IF rMesureDis[4]<rSetPoint[4]-rTolerance[4] OR rMesureDis[4]>rSetPoint[4]+rTolerance[4] THEN
bMesOutOfToler[4]:= TRUE;
ELSE
bMesOutOfToler[4]:= FALSE;	
END_IF
// Statistic ========================================
IF rMesureDis[4]<rSetPoint[4]-rTolerance[4] THEN
	stMesureStat[4].bOutLimitMin := TRUE;
ELSIF rMesureDis[4]>rSetPoint[4]+rTolerance[4] THEN
	stMesureStat[4].bOutLimitMax := TRUE;
ELSE
    stMesureStat[4].bOutLimitMin := FALSE;
    stMesureStat[4].bOutLimitMax := FALSE; 	
END_IF
//===================================================
IF bSetpChanged THEN
	nTempSeqStep:= 145;
	nMesureSeq := 150; 
END_IF
150:
IF  tonSequTim[2].Q AND rtrigSeqTrig[2].Q THEN
	// Statistic ========================================
    stMesureStat[1].bOutLimitMin := FALSE;
    stMesureStat[1].bOutLimitMax := FALSE;	
    stMesureStat[2].bOutLimitMin := FALSE;
    stMesureStat[2].bOutLimitMax := FALSE;	
    stMesureStat[3].bOutLimitMin := FALSE;
    stMesureStat[3].bOutLimitMax := FALSE;	
    stMesureStat[4].bOutLimitMin := FALSE;
    stMesureStat[4].bOutLimitMax := FALSE; 
    //===================================================
	bMesOutOfToler[1]:= FALSE;
    bMesOutOfToler[2]:= FALSE;
	bMesOutOfToler[3]:= FALSE;
	bMesOutOfToler[4]:= FALSE;
	nTempSeqStep:= 155;
	nMesureSeq := 160; 
END_IF
160:
IF bSetpChanged THEN
	nTempSeqStep:= 160;
	nMesureSeq := 10; 
END_IF
//=================================================================================================================
200: // Variable 2 choose for reference point
rMesureDis[2] := rSetPoint[2] - rMesuredValue[2]; // Diference  on Distance mesure 1
IF bSetpChanged THEN
	nTempSeqStep:= 200;
	nMesureSeq := 205; 
END_IF
205:// If it is in Tolerance
IF rMesureDis[2]<rSetPoint[2]-rTolerance[2] OR rMesureDis[2]>rSetPoint[2]+rTolerance[2] THEN
bMesOutOfToler[2]:= TRUE;
ELSE
bMesOutOfToler[2]:= FALSE;	
END_IF
// Statistic ========================================
IF rMesureDis[2]<rSetPoint[2]-rTolerance[2] THEN
	stMesureStat[2].bOutLimitMin := TRUE;
ELSIF rMesureDis[2]>rSetPoint[2]+rTolerance[2] THEN
	stMesureStat[2].bOutLimitMax := TRUE;
ELSE
    stMesureStat[2].bOutLimitMin := FALSE;
    stMesureStat[2].bOutLimitMax := FALSE; 	
END_IF
//===================================================
IF bSetpChanged THEN
	nTempSeqStep:= 205;
	nMesureSeq := 210; 
END_IF
210:// Mesure 1 value 
rMesureDis[1]:= rMesuredValue[1] - rMesuredValue[2];
IF bSetpChanged THEN
	nTempSeqStep:= 210;
	nMesureSeq := 215; 
END_IF
215:// If it is in Tolerance
IF rMesureDis[1]<rSetPoint[1]-rTolerance[1] OR rMesureDis[1]>rSetPoint[1]+rTolerance[1] THEN
bMesOutOfToler[1]:= TRUE;
ELSE
bMesOutOfToler[1]:= FALSE;	
END_IF
// Statistic ========================================
IF rMesureDis[1]<rSetPoint[1]-rTolerance[1] THEN
	stMesureStat[1].bOutLimitMin := TRUE;
ELSIF rMesureDis[1]>rSetPoint[1]+rTolerance[1] THEN
	stMesureStat[1].bOutLimitMax := TRUE;
ELSE
    stMesureStat[1].bOutLimitMin := FALSE;
    stMesureStat[1].bOutLimitMax := FALSE; 	
END_IF
//===================================================
IF bSetpChanged THEN
	nTempSeqStep:= 215;
	nMesureSeq := 220; 
END_IF
220: // Mesure 3 value 
rMesureDis[3]:= rMesuredValue[3] - rMesuredValue[2];
IF bSetpChanged THEN
	nTempSeqStep:= 220;
	nMesureSeq := 225; 
END_IF
225:// If it is in Tolerance
IF rMesureDis[3]<rSetPoint[3]-rTolerance[3] OR rMesureDis[3]>rSetPoint[3]+rTolerance[3] THEN
bMesOutOfToler[3]:= TRUE;
ELSE
bMesOutOfToler[3]:= FALSE;	
END_IF
// Statistic ========================================
IF rMesureDis[3]<rSetPoint[3]-rTolerance[3] THEN
	stMesureStat[3].bOutLimitMin := TRUE;
ELSIF rMesureDis[3]>rSetPoint[3]+rTolerance[3] THEN
	stMesureStat[3].bOutLimitMax := TRUE;
ELSE
    stMesureStat[3].bOutLimitMin := FALSE;
    stMesureStat[3].bOutLimitMax := FALSE; 	
END_IF
//===================================================
IF bSetpChanged THEN
	nTempSeqStep:= 225;
	nMesureSeq := 240; 
END_IF
240:  // Mesure 4 value 
rMesureDis[4]:= rMesuredValue[4] - rMesuredValue[2];
IF bSetpChanged THEN
	nTempSeqStep:= 240;
	nMesureSeq := 245; 
END_IF
245:// If it is in Tolerance
IF rMesureDis[4]<rSetPoint[4]-rTolerance[4] OR rMesureDis[4]>rSetPoint[4]+rTolerance[4] THEN
bMesOutOfToler[4]:= TRUE;
ELSE
bMesOutOfToler[4]:= FALSE;	
END_IF
// Statistic ========================================
IF rMesureDis[4]<rSetPoint[4]-rTolerance[4] THEN
	stMesureStat[4].bOutLimitMin := TRUE;
ELSIF rMesureDis[4]>rSetPoint[4]+rTolerance[4] THEN
	stMesureStat[4].bOutLimitMax := TRUE;
ELSE
    stMesureStat[4].bOutLimitMin := FALSE;
    stMesureStat[4].bOutLimitMax := FALSE; 	
END_IF
//===================================================
IF bSetpChanged THEN
	nTempSeqStep:= 245;
	nMesureSeq := 250; 
END_IF
250:
IF  tonSequTim[3].Q AND rtrigSeqTrig[2].Q THEN
	// Statistic ========================================
    stMesureStat[1].bOutLimitMin := FALSE;
    stMesureStat[1].bOutLimitMax := FALSE;	
    stMesureStat[2].bOutLimitMin := FALSE;
    stMesureStat[2].bOutLimitMax := FALSE;	
    stMesureStat[3].bOutLimitMin := FALSE;
    stMesureStat[3].bOutLimitMax := FALSE;	
    stMesureStat[4].bOutLimitMin := FALSE;
    stMesureStat[4].bOutLimitMax := FALSE; 
    //===================================================	
	bMesOutOfToler[1]:= FALSE;
    bMesOutOfToler[2]:= FALSE;
	bMesOutOfToler[3]:= FALSE;
	bMesOutOfToler[4]:= FALSE;
	nTempSeqStep:= 255;
	nMesureSeq := 260; 
END_IF
260:
IF bSetpChanged THEN
	nTempSeqStep:= 260;
	nMesureSeq := 10; 
END_IF
//=================================================================================================================
300: // Variable 3 choose for reference point
rMesureDis[3] := rSetPoint[3] - rMesuredValue[3]; // Diference  on Distance mesure 1
IF bSetpChanged THEN
	nTempSeqStep:= 300;
	nMesureSeq := 305; 
END_IF
305:// If it is in Tolerance
IF rMesureDis[3]<-rTolerance[3] OR rMesureDis[3]>rTolerance[3] THEN
bMesOutOfToler[3]:= TRUE;
ELSE
bMesOutOfToler[3]:= FALSE;	
END_IF
// Statistic ========================================
IF rMesureDis[3]<rSetPoint[3]-rTolerance[3] AND bMesOutOfToler[3] THEN
	stMesureStat[3].bOutLimitMin := TRUE;
ELSIF rMesureDis[3]>rSetPoint[3]+rTolerance[3] AND bMesOutOfToler[3] THEN
	stMesureStat[3].bOutLimitMax := TRUE;
ELSE
    stMesureStat[3].bOutLimitMin := FALSE;
    stMesureStat[3].bOutLimitMax := FALSE; 	
END_IF
//===================================================
IF bSetpChanged THEN
	nTempSeqStep:= 305;
	nMesureSeq := 310; 
END_IF
310:// Mesure 2 value 
rMesureDis[2]:= rMesuredValue[2]- rMesuredValue[3];    
IF bSetpChanged THEN
	nTempSeqStep:= 310;
	nMesureSeq := 315; 
END_IF
315:// If it is in Tolerance
IF rMesureDis[2]<rSetPoint[2]-rTolerance[2] OR rMesureDis[2]>rSetPoint[2]+rTolerance[2] THEN
bMesOutOfToler[2]:= TRUE;
ELSE
bMesOutOfToler[2]:= FALSE;	
END_IF
// Statistic ========================================
IF rMesureDis[2]<rSetPoint[2]-rTolerance[2] THEN
	stMesureStat[2].bOutLimitMin := TRUE;
ELSIF rMesureDis[2]>rSetPoint[2]+rTolerance[2] THEN
	stMesureStat[2].bOutLimitMax := TRUE;
ELSE
    stMesureStat[2].bOutLimitMin := FALSE;
    stMesureStat[2].bOutLimitMax := FALSE; 	
END_IF
//===================================================
IF bSetpChanged THEN
	nTempSeqStep:= 315;
	nMesureSeq := 320; 
END_IF
320: // Mesure 1 value 
rMesureDis[1]:= rMesuredValue[1] - rMesuredValue[3];
IF bSetpChanged THEN
	nTempSeqStep:= 320;
	nMesureSeq := 325; 
END_IF
325:// If it is in Tolerance
IF rMesureDis[1]<rSetPoint[1]-rTolerance[1] OR rMesureDis[1]>rSetPoint[1]+rTolerance[1] THEN
bMesOutOfToler[1]:= TRUE;
ELSE
bMesOutOfToler[1]:= FALSE;	
END_IF
// Statistic ========================================
IF rMesureDis[1]<rSetPoint[1]-rTolerance[1] THEN
	stMesureStat[1].bOutLimitMin := TRUE;
ELSIF rMesureDis[1]>rSetPoint[1]+rTolerance[1] THEN
	stMesureStat[1].bOutLimitMax := TRUE;
ELSE
    stMesureStat[1].bOutLimitMin := FALSE;
    stMesureStat[1].bOutLimitMax := FALSE; 	
END_IF
//===================================================
IF bSetpChanged THEN
	nTempSeqStep:= 325;
	nMesureSeq := 340; 
END_IF
340:  // Mesure 4 value 
rMesureDis[4]:=  rMesuredValue[4] - rMesuredValue[3];
IF bSetpChanged THEN
	nTempSeqStep:= 340;
	nMesureSeq := 345; 
END_IF
345:// If it is in Tolerance
IF rMesureDis[4]<rSetPoint[4]-rTolerance[4] OR rMesureDis[4]>rSetPoint[4]+rTolerance[4] THEN
bMesOutOfToler[4]:= TRUE;
ELSE
bMesOutOfToler[4]:= FALSE;	
END_IF
// Statistic ========================================
IF rMesureDis[4]<rSetPoint[4]-rTolerance[4] THEN
	stMesureStat[4].bOutLimitMin := TRUE;
ELSIF rMesureDis[4]>rSetPoint[4]+rTolerance[4] THEN
	stMesureStat[4].bOutLimitMax := TRUE;
ELSE
    stMesureStat[4].bOutLimitMin := FALSE;
    stMesureStat[4].bOutLimitMax := FALSE; 	
END_IF
//===================================================
IF bSetpChanged THEN
	nTempSeqStep:= 345;
	nMesureSeq := 350; 
END_IF
350:
IF tonSequTim[4].Q AND rtrigSeqTrig[2].Q THEN
	// Statistic ========================================
    stMesureStat[1].bOutLimitMin := FALSE;
    stMesureStat[1].bOutLimitMax := FALSE;	
    stMesureStat[2].bOutLimitMin := FALSE;
    stMesureStat[2].bOutLimitMax := FALSE;	
    stMesureStat[3].bOutLimitMin := FALSE;
    stMesureStat[3].bOutLimitMax := FALSE;	
    stMesureStat[4].bOutLimitMin := FALSE;
    stMesureStat[4].bOutLimitMax := FALSE; 
    //===================================================	
	bMesOutOfToler[1]:= FALSE;
    bMesOutOfToler[2]:= FALSE;
	bMesOutOfToler[3]:= FALSE;
	bMesOutOfToler[4]:= FALSE;
	nTempSeqStep:= 355;
	nMesureSeq := 360; 
END_IF
360:
IF bSetpChanged THEN
	nTempSeqStep:= 360;
	nMesureSeq := 10; 
END_IF
//=================================================================================================================
400: // Variable 4 choose for reference point
rMesureDis[4] := rSetPoint[4] - rMesuredValue[4]; // Diference  on Distance mesure 1
IF bSetpChanged THEN
	nTempSeqStep:= 400;
	nMesureSeq := 405; 
END_IF
405:// If it is in Tolerance
IF rMesureDis[4]<rSetPoint[4]-rTolerance[4] OR rMesureDis[4]>rSetPoint[4]+rTolerance[4] THEN
bMesOutOfToler[4]:= TRUE;
ELSE
bMesOutOfToler[4]:= FALSE;	
END_IF
// Statistic ========================================
IF rMesureDis[4]<rSetPoint[4]-rTolerance[4] THEN
	stMesureStat[4].bOutLimitMin := TRUE;
ELSIF rMesureDis[4]>rSetPoint[4]+rTolerance[4] THEN
	stMesureStat[4].bOutLimitMax := TRUE;
ELSE
    stMesureStat[4].bOutLimitMin := FALSE;
    stMesureStat[4].bOutLimitMax := FALSE; 	
END_IF
//===================================================
IF bSetpChanged THEN
	nTempSeqStep:= 405;
	nMesureSeq := 410; 
END_IF
410:// Mesure 2 value 
rMesureDis[2]:= rMesuredValue[2] - rMesuredValue[4];
IF bSetpChanged THEN
	nTempSeqStep:= 410;
	nMesureSeq := 415; 
END_IF
415:// If it is in Tolerance
IF rMesureDis[2]<rSetPoint[2]-rTolerance[2] OR rMesureDis[2]>rSetPoint[2]+rTolerance[2] THEN
bMesOutOfToler[2]:= TRUE;
ELSE
bMesOutOfToler[2]:= FALSE;	
END_IF
// Statistic ========================================
IF rMesureDis[2]<rSetPoint[2]-rTolerance[2] THEN
	stMesureStat[2].bOutLimitMin := TRUE;
ELSIF rMesureDis[2]>rSetPoint[2]+rTolerance[2] THEN
	stMesureStat[2].bOutLimitMax := TRUE;
ELSE
    stMesureStat[2].bOutLimitMin := FALSE;
    stMesureStat[2].bOutLimitMax := FALSE; 	
END_IF
//===================================================
IF bSetpChanged THEN
	nTempSeqStep:= 415;
	nMesureSeq := 420; 
END_IF
420: // Mesure 3 value 
rMesureDis[3]:= rMesuredValue[3] - rMesuredValue[4];
IF bSetpChanged THEN
	nTempSeqStep:= 420;
	nMesureSeq := 425; 
END_IF
425:// If it is in Tolerance
IF rMesureDis[3]<rSetPoint[3]-rTolerance[3] OR rMesureDis[3]>rSetPoint[3]+rTolerance[3] THEN
bMesOutOfToler[3]:= TRUE;
ELSE
bMesOutOfToler[3]:= FALSE;	
END_IF
// Statistic ========================================
IF rMesureDis[3]<rSetPoint[3]-rTolerance[3] THEN
	stMesureStat[3].bOutLimitMin := TRUE;
ELSIF rMesureDis[3]>rSetPoint[3]+rTolerance[3] THEN
	stMesureStat[3].bOutLimitMax := TRUE;
ELSE
    stMesureStat[3].bOutLimitMin := FALSE;
    stMesureStat[3].bOutLimitMax := FALSE; 	
END_IF
//===================================================
IF bSetpChanged THEN
	nTempSeqStep:= 425;
	nMesureSeq := 440; 
END_IF
440:  // Mesure 1 value 
rMesureDis[1]:= rMesuredValue[1] - rMesuredValue[4];
IF bSetpChanged THEN
	nTempSeqStep:= 440;
	nMesureSeq := 445; 
END_IF
445:// If it is in Tolerance
IF rMesureDis[1]<rSetPoint[1]-rTolerance[1] OR rMesureDis[1]>rSetPoint[1]+rTolerance[1] THEN
bMesOutOfToler[1]:= TRUE;
ELSE
bMesOutOfToler[1]:= FALSE;	
END_IF
// Statistic ========================================
IF rMesureDis[1]<rSetPoint[1]-rTolerance[1] THEN
	stMesureStat[1].bOutLimitMin := TRUE;
ELSIF rMesureDis[1]>rSetPoint[1]+rTolerance[1] THEN
	stMesureStat[1].bOutLimitMax := TRUE;
ELSE
    stMesureStat[1].bOutLimitMin := FALSE;
    stMesureStat[1].bOutLimitMax := FALSE; 	
END_IF
//===================================================
IF bSetpChanged THEN
	nTempSeqStep:= 445;
	nMesureSeq := 450; 
END_IF
450:
IF  tonSequTim[5].Q AND rtrigSeqTrig[2].Q THEN
	// Statistic ========================================
    stMesureStat[1].bOutLimitMin := FALSE;
    stMesureStat[1].bOutLimitMax := FALSE;	
    stMesureStat[2].bOutLimitMin := FALSE;
    stMesureStat[2].bOutLimitMax := FALSE;	
    stMesureStat[3].bOutLimitMin := FALSE;
    stMesureStat[3].bOutLimitMax := FALSE;	
    stMesureStat[4].bOutLimitMin := FALSE;
    stMesureStat[4].bOutLimitMax := FALSE; 
    //===================================================	
	bMesOutOfToler[1]:= FALSE;
    bMesOutOfToler[2]:= FALSE;
	bMesOutOfToler[3]:= FALSE;
	bMesOutOfToler[4]:= FALSE;
	nTempSeqStep:= 155;
	nMesureSeq := 160; 
END_IF
460:
IF bSetpChanged THEN
	nTempSeqStep:= 460;
	nMesureSeq := 10; 
END_IF
//=================================================================================================================
500: // Allarm on Mesure 
bMesFuncFault := TRUE;
IF tonSequTim[1].Q THEN
   nMesureSeq := 510;
END_IF
510:
bMesFuncFault := FALSE;
IF NOT bMesFuncFault THEN
	nMesureSeq := 10;
END_IF
	
END_CASE

END_FUNCTION_BLOCK

// ---- POUs/G_Utility/FB_TerminalInfo.TcPOU
FUNCTION_BLOCK FB_TerminalInfo
VAR_INPUT
	nTerminalState  : UINT;
END_VAR
VAR_OUTPUT
	sTerminalState  : STRING;
END_VAR
VAR
END_VAR

IF nTerminalState = 1 THEN 
   sTerminalState := 'Initialization';
ELSIF  nTerminalState = 2 THEN 
   sTerminalState := 'PREOP';  
ELSIF  nTerminalState = 3 THEN 
   sTerminalState := 'BOOT'; 
ELSIF  nTerminalState = 4 THEN 
   sTerminalState := 'SAFEOP';   
ELSIF  nTerminalState = 8 THEN 
   sTerminalState := 'OPERATIONAL';
ELSIF  nTerminalState = 16#0010 THEN 
   sTerminalState := 'Slave signals error';   
ELSIF  nTerminalState = 16#0020 THEN 
   sTerminalState := 'Invalid vendorId, productCode... read';  
ELSIF  nTerminalState = 16#0040 THEN 
   sTerminalState := 'Initialization error occurred';   
ELSIF  nTerminalState = 16#0080 THEN 
   sTerminalState := 'Slave disabled';   
ELSIF  nTerminalState = 16#0100 THEN 
   sTerminalState := 'Slave not present';    
ELSIF  nTerminalState = 16#0200 THEN 
   sTerminalState := 'Slave signals link error';    
ELSIF  nTerminalState = 16#0400 THEN 
   sTerminalState := 'Slave signals missing link'; 
ELSIF  nTerminalState = 16#0800 THEN 
   sTerminalState := 'Slave signals unexpected link';
ELSIF  nTerminalState = 16#1000 THEN 
   sTerminalState := 'Communication port A';
ELSIF  nTerminalState = 16#2000 THEN 
   sTerminalState := 'Communication port B';
ELSIF  nTerminalState = 16#4000 THEN 
   sTerminalState := 'Communication port C';
ELSIF  nTerminalState = 16#8000 THEN 
   sTerminalState := 'Communication port D'; 	
END_IF

END_FUNCTION_BLOCK
